(* CoDeSys 2.3 project: cy-162.pro *)
(* Title: cy-wg-24 - ClevergyAS *)
(* Author: Andrea Laini *)
(* Libraries: OSCAT\oscat_basic_333_pfc_2000.lib*20.4.16 13:29:42, mod_com.lib 16.5.13 14:00:50, SerComm.lib 16.5.13 14:00:50, Serial_Interface_01.lib 22.4.13 12:50:14, Modb_l05.lib*22.4.13 12:50:12, SysLibFile.lib 16.5.13 14:00:50, Util.lib 16.5.13 14:00:50, SYSLIBCALLBACK.LIB 16.5.13 14:00:50, SysLibRtc.lib 16.5.13 14:00:50, SysLibSockets.lib 22.5.14 16:16:32, SysLibEvent.lib 16.5.13 14:00:50, SysLibTime.lib 16.5.13 14:00:48, SysLibPlcCtrl.lib 16.5.13 14:00:50, SysLibStr.lib 16.5.13 14:00:50, Standard.lib 20.5.14 08:13:26, Iecsfc.lib 16.5.13 14:00:50 *)

(* PLC configuration (modules and I/O channels)
VPN_STATUS AT %IX0.0 [BOOLOnX_I] I 1: Digital Input
DI02 AT %IX0.1 [BOOLOnX_I] I 2: Digital Input
COORD_STATUS AT %IX0.2 [BOOLOnX_I] I 3: Digital Input
DI04 AT %IX0.3 [BOOLOnX_I] I 4: Digital Input
Modbus variables [PFC200MODBUS] node 1, in %IB0 out %QB0 {PlcStopBehaviour = 1; FiledbusErrorBehaviour = 1; TcpOperation = 0; TcpPort = 502; TcpTimeout = 600; UdpOperation = 0; UdpPort = 502; RtuOperation = 0; NodeId = 200; ResponseTimeout = 5000; Interface = 0; Baud = 38400; StopBits = 2; Parity = 0; FlowCtrl = 0; PhysInterface = 1}
Modbus-Master [MB_MASTER] node 2, in %IB0 out %QB0
*)

(* Global variable list: Global_Constants *)
VAR_GLOBAL CONSTANT

	Plant_NAME			: STRING :='cySN:162  cyVER:0 Q5904 via COMBONI Desenzano';
	Plant_SN				: DWORD  :=162;	  	(* S/N Impianto di telecontrollo *)
	Plant_SW_VER			: WORD   :=0;		(* Versione SW installata *)


	GEOLUMEN_COORD_VERSION:BYTE:=2;


	(* Plant-dependent constants *)
	LATITUDE 										: REAL:=45.45522;
	LONGITUDE										: REAL:=10.56686;
	ASTRO_TWILIGHT_MORNING_MODE					: BYTE:=0;
	ASTRO_TWILIGHT_EVENING_MODE					: BYTE:=0;
	COUNTRY_CODE 									: STRING:='IT';
	MAX_LUXNUM										: WORD := 1;
	MAX_GEOLUMENNODES								: WORD :=MAX_LUXNUM;
	MAX_LOG_ROW									: WORD :=2; (*MAX_LUXNUM	/10 +1 per eccesso*)
	MAX_RETRY_NO_FEEDBACK_GEOLUMEN_NODES			: WORD:=20;
	MAX_RETRY_STATUS_NOT_ALIGNED_GEOLUMEN_NODES       : WORD:=360;
	TIME_WAIT_RETRY_NOT_ALIGNED						: TIME:=T#10m;
	TIME_NO_FEEBACK_RESEND_STATUS					: TIME:=T#20m;

	(*tempi debug comandi global *)
	PRE_TIME_ENFORCE_GON 							: TIME:=T#10m;
	PRE_TIME_CLOSE_GOFF 								: TIME:=T#100m;
	TRIALS_ENFORCE_GON 								: WORD:=60;
	PERIOD_ENFORCE_GON 								: TIME:=T#1m;
	PERIOD_ENFORCE_GOFF 							: TIME:=T#15m;

	GEOLUMEN_SEND_TIME : TIME:=T#1s;

	(* Internal, tech const *)
	MAX_ARRAY_MSG	: BYTE:=250;
	ANALOG			: BOOL:=0;
	DIGITAL			: BOOL:=1;

	(* Filesystem *)
	FilesPath  			: STRING :='/media/sd/';
	MapConf_Path			: STRING :=	'/media/sd/';

	Luxlist_FileName	: STRING :='_LUX_LIST.txt';
	Cfg_FileName		: STRING :='CFG.txt';

	(* Colour Visu *)
	COLOR_RED			: DWORD 	:= 16#2020F0;
	COLOR_YELLOW		: DWORD	:= 16#20F0F0;
	COLOR_GREEN		: DWORD	:= 16#20F020;
	COLOR_GREEN_OFF	 : DWORD	:= 16#108010;

	(* TCP Logger *)
	Logger_SERVER		: STRING:='';
	Logger_IP				: STRING:='192.168.100.3';
	Logger_PORT			: WORD  :=80;
	Logger_GETSTART		: STRING:='GET /cygmsrv/hsgm.ashx?';
	Logger_GETEND		: STRING:='$R$N$R$N';
	Logger_CHECK			: STRING:='True';
	Logger_CRLF			: STRING:='$R$N';
	Logger_DataFile		: STRING:='/media/sd/LOG.DAT';
	Logger_DataFileOld	: STRING:='/media/sd/LOG.BCK';
	Logger_IndexFile	: STRING:='/media/sd/LOG.IDX';
	Logger_ConnRetries	: BYTE:=5;
	Logger_RecoverMsgs	: BYTE:=25;

	(* TCP Remote *)
	Remote_PORT			: WORD  :=10;
	Remote_WELCOME		: STRING:='Connected$R$N';
	Remote_OK			: STRING:='OK$R$N';
	Remote_ERROR		: STRING:='ERROR$R$N';

	(* TCP Sockets *)
	MAX_SEND_TCP_SERVER					 : DWORD:=6000;(*60000*)
	MAX_RECEIVE_TCP_SERVER				 : DWORD:=12000;
	MAX_RECEIVE_TCP_SERVER_SOCKET	 	 : DWORD:=6000;
	MAX_SEND_TCP_CLIENT					 : DWORD:=6000;(*15000*)
	MAX_RECEIVE_TCP_CLIENT				 : DWORD:=6000;
	MAX_RECEIVE_TCP_CLIENT_SOCKET		 : DWORD:=6000;
	MAX_RECEIVE_UDP_SERVER				 : INT  :=1472;
	MAX_RECEIVE_UDP_CLIENT				 : INT  :=1472;
	CONNECT_WATCHDOG_TIME				 : TIME :=t#10s;


END_VAR

(* Global variable list: Global_Retain *)
VAR_GLOBAL RETAIN PERSISTENT

	(* valori retain per i LUX objects*)
	GlobalWorkingtime		: ARRAY [1..MAX_LUXNUM] OF DWORD; (* [sec] Internal working time counter *)
	GlobalPowerOnCycles	: ARRAY [1..MAX_LUXNUM] OF WORD;	(*/DWORD;  *) (* Internal counter of power-on cycles *)
	GlobalEnergyCounter	: ARRAY [1..MAX_LUXNUM] OF WORD; (* DWORD;  *) (* [E-1 kWh] Internal energy counter *)
	GlobalEnergyCounter_t 	: ARRAY [1..MAX_LUXNUM] OF DWORD; (* Temporary energy in E-2*Wsec *)

	(*configurazione degli astro *)
	ASTR_CONFIG   : ARRAY [1..MAX_LUXNUM] OF  type_ASTR_config;

	USE_RETAIN:BOOL:=FALSE;

	DEBUG_NO_CONTROL_LIGHTS : BOOL :=FALSE;
	DEBUG_SERIAL:BOOL:=FALSE;
	DEBUG_SAVE_SNAPSHOT:BOOL:=TRUE;
	USING_EXTERNAL_ASTRO:BOOL:=TRUE;

END_VAR

(* Global variable list: Global_Variables *)
VAR_GLOBAL

	SYS    : typ_SYS;
	Logger : typ_Logger;

	LAMP : LAMP_AL_GENERALE;

	PLC_ID				: STRING:='1' ; (* Identificativo del plc - interno al file cfg.txt  *)
	PLC_START_TIME 		:DT;

	SyncLogRequest: BOOL:=FALSE;
	TimerLogLux : ARRAY[1..MAX_LOG_ROW] OF TON;
	TimerLogLuxSync : ARRAY[1..MAX_LOG_ROW] OF TON;
	TimerLogLuxSyncDone : ARRAY[1..MAX_LOG_ROW] OF BOOL;
	TimingLuxBase : TIME;
	logRowLux:INT:=0;
	IS_PRE_GLOBAL_ON_ONGOING:BOOL:=FALSE;

	(*contSts0:DWORD:=0;
	contSts1:DWORD:=0;*)
	warningHFileLogSend:BOOL:=FALSE;

	(*Tabella della lista dei lux GEOLUMEN costruita sulla base del file di configurazione*)
	TabListLux : ARRAY [1..MAX_LUXNUM] OF type_TabListLuxGeolumen;
	TabListLuxSendAuth : ARRAY [1..MAX_LUXNUM]  OF WORD:=0;

	LuxElement		: ARRAY [1..MAX_LUXNUM] OF obj_LUX:=(CTRL_MODE:=2,CTRL_MODE_BackUp:=2); (* Lista di variabili Lux   *)
	LuxGeolumenChangeFlag : ARRAY [1..MAX_LUXNUM] OF INT;

	TimerLogAstro : ARRAY[1..MAX_LOG_ROW] OF TON;
	TimerLogAstroSync : ARRAY[1..MAX_LOG_ROW] OF TON;
	TimerLogAstroSyncDone : ARRAY[1..MAX_LOG_ROW] OF BOOL;
	TimingAstroBase : TIME;
	tIndex:INT;
	logRowAstro:INT:=0;
	isGeolumenNodesOffDuringDay:isGeolumenNodesOffDuringDay;
	tmpBoolGoffDay:BOOL;

	GeolumenNodeList	:GeolumenNodeList;

	(* Astro crono *)
	ASTR   			: ARRAY [1..MAX_LUXNUM] OF obj_ASTR;
	astroGen			 : obj_ASTR;
	CronEd : obj_CRON_EDITOR:=(crono_type:='ASTR');

	(*Lux *)
	MsgRecBuffer	: ARRAY[0..MAX_ARRAY_MSG ] OF type_MsgReceive; (*Array contenente i messaggi in arrivo e gestito in modo circolare*)
	KEYON :BOOL;

	LuxGeolumenNodes : ARRAY [1..MAX_LUXNUM] OF obj_GeolumenNode:=(MAX_RETRY_NO_FEEDBACK:=MAX_RETRY_NO_FEEDBACK_GEOLUMEN_NODES,
															MAX_RETRY_STATUS_NOT_ALIGNED:=MAX_RETRY_STATUS_NOT_ALIGNED_GEOLUMEN_NODES);

	LuxGeolumenNodesAlignFlags : ARRAY [1..MAX_LUXNUM] OF BOOL:=FALSE;
	LuxGeolumenNodesCurrent : ARRAY [1..MAX_LUXNUM] OF DWORD;
	Missing : ARRAY [1..MAX_LUXNUM] OF BOOL:=FALSE;
	missingCount:INT:=0;

	(*Geolumen rs232 dependent*)
	COM0:SERIAL_INTERFACE := (xOPEN_COM_PORT := TRUE, bCOM_PORT_NR  := 0, cbsBYTESIZE := BS_8,
							cbBAUDRATE := BAUD_115200, cpPARITY := PARITY_NO, csSTOPBITS := STOPBITS_1, cfFLOW_CONTROL := NO_FLOW_CONTROL);
	ReceiveBuffer:typRing_Buffer;
	xCoupledAll		:BOOL;
	obj_GeolumenCoordinator:obj_GeolumenCoordinator;
	LuxGeolumenDiagnostics:LuxGeolumenDiagnostics;
	SendDataQueue:SendDataQueue;

END_VAR

(* Data type in DT_LUX *)
TYPE en_ActionKey :
(
	NormalMode 	:= 0,
	SwitchON		:= 1,
	SwitchOFF		:= 2,
	Restore			:= 3
);
END_TYPE

(* Data type in DT_LUX *)
TYPE en_KeyMode :
(
	BUTTON_NO		:=01,
	BUTTON_NC		:=02,
	SWITCH_NO		:=03,
	SWITCH_NC			:=04
);
END_TYPE

(* Data type in DT_Logger *)
TYPE en_Logger_ErrLev :
(
	EL_Log			:=0,
	EL_Wrn			:=1,
	EL_Alarm		:=2,
	EL_AlarmStop	:=3,

	EL_Evt			:=4
);
END_TYPE

(* Data type in DT_Logger *)
TYPE en_Logger_Status :
(
	S_Logger_UNKNOWN := 0,
	S_Logger_IDLE,
	S_Logger_WAITCONN,
	S_Logger_WAITTX,
	S_Logger_WAITRESP,
	S_Logger_ERROR
);
END_TYPE

(* Data type in DT_LUX *)
TYPE en_Modality :
(
	ManualeOff 	:= 0,
	ManualeOn 	:= 1,
	Cronografo	:= 2,
	Timer		:= 3,
	KeyControl	:= 4
);
END_TYPE

(* Data type in System *)
TYPE en_MsgType :
(
	COMPLETED:=0, (*Il messaggio è stato elaborato*)
	REQAUTH0:= 1,  (*Richiesta in corso a cui rispondere*)
	REQAUTH1:=2,  (*Nodo già acquisito in rete*)
	DATAREC:=3,
	ECHO:=4,
	NODE_DELETED:=5,
	MED:=6
);
END_TYPE

(* Data type in System *)
TYPE en_StartingState :
(
	NOT_AUTHORISE  := 0,
	READ_NODE
);
END_TYPE

(* Data type in DT_SYS *)
TYPE en_SYS_Objects :
(
	EO_SYS		:=0,  (* PLC *)
	EO_VPN		:=1,  (* VPN *)
	EO_DOOR	:=2,  (* Door & access control *)

	EO_CAL		:=10, (* Caldaia *)
	EO_CIR		:=11, (* Circolatore *)
	EO_CRON		:=12, (* Crono-termostato *)
	EO_VRD		:=13, (* Valvola miscelatore pannelli *)
	EO_CTL		:=14, (* Contalitri *)
	EO_CTB		:=15, (* Contabilizzatore *)
	EO_TPV		:=16, (* Temperature probes values *)
	EO_PPV		:=17, (* Pressure probes values *)
	EO_PBV		:=18, (* Over-Pressure Alarms *)
	EO_TBV		:=19, (* Over-Temperature Alarms *)
	EO_PMV		:=20, (* Under-Pressure Alarms *)
	EO_GRU		:=21, (* Gruppo termico *)
	EO_PDC		:=22, (* Pompa di calore *)
	EO_SOL		:=23, (* Pannello solare termico *)
	EO_ESOL		:=24, (* Pannello solare fotovoltaico *)
	EO_GAS		:=25, (* Contatore GAS *)
	EO_PORT		:=26, (* Misuratore di portata *)
	EO_FPV		:=27, (* Flow probes values *)
	EO_ANZ		:=28, (* Analizzatore di rete *)
	EO_SCA		:=29, (* Signal Control Alarms *)
	EO_LUX		:=30, (* Illumination point *)
	EO_LUXM		:=31, (* Metered illumination point*)
	EO_PSG		:=32, (* Sensore di passaggio *)
	EO_HVAC		:=33, (*Heating, Ventilating and Air Conditioning*)
	EO_HYGRV	:=34, (*Valori sensori di umidità relativa (0.1%)*)
	EO_COOV		:=35, (*Valori sensori CO2 (PPM)*)

	EO_ASTR		 :=46, (*Astro crono *)




	EO_ZGW			:=200,  (* ZigBee - Gateway *)
	EO_ZRM			:=201,	(* ZigBee - Repeater *)
	EO_ZREL			:=202,	(* ZigBee - Actuator rele *)
	EO_ZTHL			:=203,	(* ZigBee - Temperature Sensor *)

	EO_ASGW			:=250,	(* ASi - Gateway *)
	EO_ASCBI			:=251,	(* ASi - Input Board, Ciabatta *)

	EO_LON				:=1000, (* Bus - LON *)
	EO_MODBUS			:=1001, (* Bus - MODBUS *)
	EO_MBUS				:=1002, (* Bus - M-BUS *)
	EO_MODBUS_TCP	:=1003, (* Bus - MODBUS TCP *)

	EO_GENERIC			:=9000, (* Generic dataset *)
	EO_EXPO				:=9001 (* EXPO dataset *)
);
END_TYPE

(* Data type in DT_SYS *)
TYPE en_SYS_Status :
(
	S_UNKNOWN  := 0,
	S_STARTUP,
	S_INIT_RTC,
	S_INIT_VAR,
	S_AUTOTEST,
	S_RUNNING,
	S_SHUTDOWN,
	S_HALT,
	S_RELOAD,
	S_STARTER
);
END_TYPE

(* Data type in DT_SYS *)
TYPE typ_Condition :
STRUCT
	Enable		:	BYTE;	(*	0: Condition event not used		(disable condition event)
								1: Boolean event: trig On	(rele, switch, sensors digital input..)
								2:    ''    ''  : trig Off		
								3:	  ''    ''  : trig On/Off
								4: Tod event: trig On		(Time of day)
								5: Tod event: trig Off		(Trig On/Off not expected -> it's a schedule! )
							 *)

	(* Boolean event *)
	OnIN		:	BOOL;	(* Input event generating an On *)
	OffIN		:	BOOL;	(* Input event generating an Off  *)

	OnValue		:	BOOL;	(* Value to trig an On *)
	OffValue	:	BOOL;	(*   ''        ''   Off	 *)


	(* Time of the day event (absolute time) *)
	OnTime		:	TOD;	(* Time at which trig an On (hh:mm) *)
	OffTime		:	TOD;	(*  ''            ''     Off (hh:mm)  *)


END_STRUCT
END_TYPE

(* Data type in DT_CRON *)
TYPE typ_Cron_Calendar :
STRUCT
	Profile		: ARRAY[0..384] OF BYTE;
END_STRUCT
END_TYPE

(* Data type in DT_CRON *)
TYPE typ_Cron_Jolly :
STRUCT
	Start		: DT;
	End			: DT;
	Temp		: WORD;
	Flags		: WORD; (* B0:Enabled B1..B15:Unused *)
END_STRUCT
END_TYPE

(* Data type in DT_CRON *)
TYPE typ_Cron_Profile :
STRUCT
	Flags		: WORD;
	Setpoint	: ARRAY [0..95] OF WORD;
END_STRUCT
END_TYPE

(* Data type in DT_Logger *)
TYPE typ_Logger :
STRUCT
	Status		: en_Logger_Status;

	SendReq		: BOOL;
	SendIdx		: DWORD;
	SendData	: ARRAY [0..MAX_SEND_TCP_CLIENT] OF BYTE;
	SendLen		: DINT;

	TData		: ARRAY [0..MAX_SEND_TCP_CLIENT] OF BYTE;
	TLen		: DINT;

	LastIdxPos	: DWORD;

	(* Temporary variables used by objects *)
	s1			: STRING(256);
	i1			: WORD;

END_STRUCT
END_TYPE

(* Data type in DT_SYS *)
TYPE typ_SYS :
STRUCT
	Status			: en_SYS_Status;
	Warning		: BOOL;
	Alarm			: BOOL;
	AlarmStop		: BOOL;

	Time_LogString	: STRING(255);
	Time_Year		: WORD;
	Time_Month		: BYTE;
	Time_Day		: BYTE;
	Time_Hour		: BYTE;
	Time_Min		: BYTE;

	Time_CT_DT		: DT;
	Time_CT_Day		: WORD;
	Time_CT_Quarter	: BYTE;

	LastLogs_Idx	: BYTE;
	LastLogs_Dat	: ARRAY[0..5] OF STRING(255);
	LastLogs_Msg	: ARRAY[0..5] OF STRING(255);

END_STRUCT
END_TYPE

(* Data type *)
TYPE type_ASTR_config :
STRUCT
	id:DWORD;
	twilightMorningMode:BYTE;
	twilightEveningMode:BYTE;
	preSunrise:BYTE;
	postSunrise:BYTE;
	preSunset:BYTE;
	postSunset:BYTE;
END_STRUCT
END_TYPE

(* Data type in DT_LUX *)
(* La seguente struttura ha la funzione di collegare l'id del lux con i relativi dati qui indicati *)
(* In tal modo la visualizzazione dello stato dei lux viene eseguita associando l'ID dell'array contenente questa struttura*)

TYPE type_DataLuxForVis :
STRUCT
	VisStatus	: DWORD; (* valori di status_vis   *)
	VisTimer	: TIME;	(* Valori dei timer  *)
	VisMod		: en_Modality; (* Impostazione mode  *)
END_STRUCT
END_TYPE

(* Data type in DT_LUX_GEOLUMEN *)
TYPE type_LuxGeolumenStatus :
STRUCT
	ID_Geolumen: DWORD;
	DimmValue_0 : WORD;
	DimmValue_1 : WORD;
	DimmValue_2 : WORD;
	LampCurrent:DWORD;LampPower:DWORD;LampVoltage:DWORD;
	lqiLast, lqiAvg, lqiMax, lqiMin:WORD;
	lastPar:STRING(255);
END_STRUCT
END_TYPE

(* Data type in DT_LUX *)
TYPE type_LuxOutput :
STRUCT
	DigitalOut	:	BOOL;
	AnalogOut	:	WORD;
	TypeOut	:	BOOL;
END_STRUCT
END_TYPE

(* Data type in System *)
TYPE type_MsgReceive :
STRUCT
	Msg		:STRING (255);
	MsgType	: en_MsgType; (*Indica il tipo di messaggio STS0, STS1,...*)
	dwMacAdd	: DWORD;

END_STRUCT
END_TYPE

(* Data type in DT_LUX *)
(* Struttura utile per la lista dei lux *)

TYPE type_TabListLux :
STRUCT
	LuxNumber: WORD;
	MODE: WORD;
	MacAdd: DWORD;
	MacAddH: WORD;
	MacAddL: WORD;
	StMacAdd	: STRING(8);
END_STRUCT
END_TYPE

(* Data type in DT_LUX_GEOLUMEN *)
(* Struttura utile per la lista dei lux *)

TYPE type_TabListLuxGeolumen :
STRUCT
	LuxNumber	: DWORD;
	LuxID_Geolumen		: DWORD;
	MacAdd	: DWORD;
	MacAddH	: WORD;
	MacAddL	: WORD;
	StMacAdd	: STRING(8);
	xCoupled	: BOOL;
END_STRUCT
END_TYPE

(* POU PLC_PRG, ST *)
PROGRAM PLC_PRG
VAR CONSTANT
	TIME_LUX_LOG_NORMAL:TIME:=T#5m;
	TIME_ASTRO_LOG_NORMAL:TIME:=T#30m;
	TIME_LUX_PROC:TIME:=T#200ms;
	TIME_STATUS_2:TIME:=T#180M;
END_VAR
VAR
	DAILY_RESET_DONE:BOOL;
	TimerLux:TON;
	Timer1: TON;  (*Fast controls tick *)
  	Timer2: TON; (* Plant control tick *)
	TimerSnapshot:TON;
	maxLoggerRow:INT;
	TimerAstroQuadroNotte:TON;
	TimerAstroQuadroGiorno:TON;
	contaSera:INT:=0;
	contaMattina:INT:=0;

	xOpenPort		: BOOL := TRUE;
	xInitPort			: BOOL;
	xSendActive	: BOOL;
	SendString		: STRING(255) := 'CMD_AUTHORISE=0';
	xStartSend		: BOOL;

	GeoNodeIndex:INT:=1;
	i :INT :=1;
	LuxCount	: WORD:=1;
	ValInCrono	: INT; (* Valore del setpoint del crono *)
	counter		: WORD;
	tmpIndex:INT;

	tmpMaxEvening:BYTE;
	tmpMinEvening:BYTE;
	tmpMinMorning:BYTE;
	tmpMinPreEvening:BYTE;
	tmpMaxPreEvening:BYTE;
	tmpMaxPostEvening:BYTE;
	tmpMinPostEvening:BYTE;
	tmpMinPreMorning:BYTE;
	tmpMaxPostMorning:BYTE;
	tmpTime:TIME;


END_VAR
(*
	Network setup:
		IP  = 192.168.100.2 | MSK = 255.255.255.0
		GW	= 192.168.100.1 | DNS = 192.168.100.1
		SNTP = 193.204.114.232 (3600s) ==> 192.168.100.3
*)


(*==============================*)
(*=====    Main control machine    ====*)
(*==============================*)

MainCtrl();

Logger_Proc();

Remote_Proc();
END_PROGRAM
ACTION MainCtrl:
CASE Sys.Status OF

	(* stato STARTUP
	     - carico la lista dei nodi Geolumen da accettare (ID palo, MAC)
	     - apro la porta seriale
	     - invio al coordinatore Geolumen il comando CMD_AUTHORISE=0
	*)
	S_STARTUP:

		DAILY_RESET_DONE:=FALSE;

		(* pongo a zero valore variabili essenziali*)
		FOR counter := 1 TO MAX_LUXNUM DO
			TabListLux[counter].LuxID_Geolumen:=0;
			TabListLux[counter].MacAdd:=0;
			TabListLux[counter].MacAddH:=0;
			TabListLux[counter].MacAddL:=0;
			TabListLux[counter].StMacAdd:='';
			TabListLux[counter].LuxNumber:=0;
			TabListLux[counter].xCoupled:=FALSE;
			LuxElement[counter].ID:=0;
			ASTR[counter].ID:=0;
			LuxGeolumenNodes[counter].ID_Lux:=0;
			LuxGeolumenNodes[counter].ID_Geolumen:=0;
		END_FOR

		(* caricamento lista nodi *)
		GeolumenNodeList();

		(* apro la porta seriale *)
		xSendActive:=FALSE;
		COM0((*	bCOM_PORT_NR 	:= 0,
				cbBAUDRATE     	 := BAUD_38400,
			(*	cbBAUDRATE 		:= wBaudRate, *)
				cbsBYTESIZE		:= BS_8,  (*bDataBits,*)
				cpPARITY			:= PARITY_NO, (* bParity,*)
				csSTOPBITS		:= STOPBITS_1,
				cfFLOW_CONTROL	:= NO_FLOW_CONTROL,	(*bFlowControl,			*) *)
				cbBAUDRATE     	 := BAUD_115200,
				utRECEIVE_BUFFER := ReceiveBuffer,
				ptSEND_BUFFER	:= ADR(SendString),
				xINIT				:=  xInitPort,
		     		xOPEN_COM_PORT 	:= TRUE,	(*xOpenPort,*)
				iBYTES_TO_SEND	:= LEN(SendString)+1,
				xSTART_SEND		:= xSendActive );

		(*proseguo con lo stato successivo sse porta seriale aperta *)
		IF COM0.xCOM_PORT_IS_OPEN THEN
			Sys.Status:=S_INIT_RTC;

			(* anzitutto blocco auto-auth da parte dei nodi*)
			obj_GeolumenCoordinator.blockNodeAutoAdd();

		END_IF

	(* stato INIT_RTC
	     - init RTC PLC
	     - sync time coordinatore Geolumen
	*)
	S_INIT_RTC:

		(* aggiorno stringhe RTC as usual*)
		RTC_Update();

		(* aggiorno ora del coordinatore con la mia e proseguo allo stato successivo come al solito *)
		IF Sys.Time_Year>2000 THEN
			obj_GeolumenCoordinator.updateNetworkTime();
			Sys.Status:=S_INIT_VAR;
		END_IF

	(* stato S_INIT_VAR
	     - init variabili oggetti
	*)
	S_INIT_VAR:

		(*tutti i LUX presenti sono di default e ad ogni riavvio di tipo dimming e di modo 2 - Cronografo *)
		FOR counter := 1 TO MAX_LUXNUM DO
			LuxElement[counter].DimmingType:=1;
			LuxElement[counter].CTRL_MODE := 2 ; (* TabDefaultLux[counter].Mode; //copio il mode nella tabella delle variabili dei lux 	*)
			LuxElement[counter].CTRL_MODE_backUp := 2;  (* TabDefaultLux[counter].Mode; //salvo il mode di backup per il ripristina modo	*)
		END_FOR

		(*ripeto il comando di esclusione di accesso da parte dei nodi, per sicurezza*)
		obj_GeolumenCoordinator.blockNodeAutoAdd();


		(* definizione ASTRO di quadro, per test *)
		tmpMinEvening:=100;
		tmpMaxEvening:=0;
		tmpMinMorning:=100;
		tmpMinPreEvening:=30;
		tmpMaxPreEvening:=0;
		tmpMaxPostEvening:=0;
		tmpMinPostEvening:=100;
		tmpMinPreMorning:=30;
		tmpMaxPostMorning:=0;

		(* inizializzo gli astro con eventale stato retain *)
		FOR i:=1 TO MAX_LUXNUM DO
			ASTR[i].ID:=ASTR_CONFIG[i].ID;
			ASTR[i].rLatitude:=LATITUDE;
			ASTR[i].rLongitude:=LONGITUDE;
			ASTR[i].countryCode:=COUNTRY_CODE;
			IF(USE_RETAIN=FALSE) THEN
				ASTR[i].twilightEveningMode :=ASTRO_TWILIGHT_EVENING_MODE;
				ASTR[i].twilightMorningMode :=ASTRO_TWILIGHT_MORNING_MODE;
				ASTR_CONFIG[i].preSunrise:=ASTR[i].preSunrise;
				ASTR_CONFIG[i].postSunrise:=ASTR[i].postSunrise;
				ASTR_CONFIG[i].preSunset:=ASTR[i].preSunset;
				ASTR_CONFIG[i].postSunset:=ASTR[i].postSunset;
				ASTR_CONFIG[i].twilightEveningMode:=ASTR[i].twilightEveningMode;
				ASTR_CONFIG[i].twilightMorningMode:=ASTR[i].twilightMorningMode;
			ELSE
				ASTR[i].preSunrise:=ASTR_CONFIG[i].preSunrise;
				ASTR[i].postSunrise:=ASTR_CONFIG[i].postSunrise;
				ASTR[i].preSunset:=ASTR_CONFIG[i].preSunset;
				ASTR[i].postSunset:=ASTR_CONFIG[i].postSunset;
				ASTR[i].twilightEveningMode:=ASTR_CONFIG[i].twilightEveningMode;
				ASTR[i].twilightMorningMode:=ASTR_CONFIG[i].twilightMorningMode;
			END_IF


			IF ASTR[i].twilightEveningMode < tmpMinEvening THEN tmpMinEvening:=ASTR[i].twilightEveningMode; END_IF
			IF ASTR[i].twilightMorningMode < tmpMinMorning THEN tmpMinMorning:=ASTR[i].twilightMorningMode; END_IF
			IF ASTR[i].preSunset > tmpMinPreEvening THEN tmpMaxPreEvening:=ASTR[i].preSunset; END_IF
			IF ASTR[i].postSunset < tmpMinPostEvening THEN tmpMinPostEvening:=ASTR[i].postSunset; END_IF
			IF ASTR[i].preSunrise < tmpMinPreMorning THEN tmpMinPreMorning:=ASTR[i].preSunrise; END_IF
			IF ASTR[i].postSunrise > tmpMaxPostMorning THEN tmpMaxPostMorning:=ASTR[i].postSunrise; END_IF

		END_FOR

		astroGen.ID:=1;
		astroGen.rLatitude:=LATITUDE;
		astroGen.rLongitude:=LONGITUDE;
		astroGen.countryCode:=COUNTRY_CODE;
		astroGen.twilightEveningMode:=tmpMinEvening;
		astroGen.twilightMorningMode:=tmpMinMorning;
		astroGen.preSunset:= tmpMaxPreEvening;
		astroGen.postSunset:= tmpMinPostEvening;
		astroGen.preSunrise:= tmpMinPreMorning;
		astroGen.postSunrise:=tmpMaxPostMorning;

		(*chiedo agli eventuali nodi geoluem connesso il loro stato*)
		SendDataQueue(pTxData:=ADR(obj_GeolumenCoordinator.getStatusAllFeedback));
		SendDataQueue.addMessage();

		(*recall lux*)
		obj_GeolumenCoordinator.luxRecall();


		(*procedo con stato successivo *)
		Sys.Status:=S_STARTER;

	(* stato S_STARTER
	     - ad oggi logga solo avvio
	*)
	S_STARTER:
		LogEv(EL_Wrn,EO_SYS,0,1,CONCAT('System_startup_v',WORD_TO_STRING(Plant_SW_VER)));
		Sys.Status:=S_RUNNING;
		PLC_START_TIME:=SYS.Time_CT_DT;

	(* stato S_RUNNING
	     - aggiorna lo stato di ASTR e di LUX
	     - si occupa di mantenere la corrispondenza di stato tra LUX e GEOLUMENNODE
	*)
	S_RUNNING:

		(*salvo stato nodi su sd, ogni ora *)
		TimerSnapshot(IN:=NOT TimerSnapshot.Q,PT:=T#1h);
		IF DEBUG_SAVE_SNAPSHOT AND TimerSnapshot.Q THEN
			GeolumenSaveNodeStatus();
		END_IF

		(*aggiorni eventi SCA e SYS as usual*)
		Timer1(IN:=NOT Timer1.Q,PT:=T#50ms);
		IF Timer1.Q THEN
			(* Update meters *)
			SCA_Proc();
			(* Update system checks *)
			SYS_Proc();
		END_IF

		(*aggiorno stringhe RTC as usual*)
		Timer2(IN:=NOT Timer2.Q,PT:=T#500ms);
		IF Timer2.Q THEN
			(* Read current date/time *)
			RTC_Update();
			(*per PIANO C*)
			isGeolumenNodesOffDuringDay(isGeolumenNodesOffDuringDay=>tmpBoolGoffDay);
		END_IF

		(* gestione astr di quadro per eventuali comandi global di enforcing e gestione PIANO C*)
		(* + reset coordinatore prima di accensione serale*)
		AstroGen(localTime:=Sys.Time_CT_DT);
		IF(SYS.Time_CT_DT>=AstroGen.timeStart-PRE_TIME_ENFORCE_GON AND SYS.Time_CT_DT<AstroGen.timeStart) THEN
			IS_PRE_GLOBAL_ON_ONGOING:=TRUE;

			FOR GeoNodeIndex:=1 TO MAX_LUXNUM  DO
				IF LuxElement[GeoNodeIndex].ID <> 0 THEN
					LuxGeolumenNodes[GeoNodeIndex].resetLampIndicators();
				END_IF
			END_FOR

		ELSE
			IS_PRE_GLOBAL_ON_ONGOING:=FALSE;
			DAILY_RESET_DONE:=FALSE;
		END_IF


		IF(IS_PRE_GLOBAL_ON_ONGOING AND DAILY_RESET_DONE=FALSE) THEN
			(*LuxGeolumenDiagnostics.executeCommandReset();*)
			DAILY_RESET_DONE:=TRUE;
		END_IF


		(* gestione con global, debug and test *)
		(*TimerAstroQuadroNotte(IN:=NOT TimerAstroQuadroNotte.Q,PT:=PERIOD_ENFORCE_GON);
		(* la sera lancio un set iniziale di Global a 100 *)
		IF(SYS.Time_CT_DT>=AstroGen.timeStart-PRE_TIME_ENFORCE_GON AND TimerAstroQuadroNotte.Q AND contaSera<TRIALS_ENFORCE_GON ) THEN
			(*obj_GeolumenCoordinator.sendGlobalON();*)(*DIEGO REMOVE*)
			contaSera:=contaSera+1;
			contaMattina:=0;
		ELSIF contaSera>=TRIALS_ENFORCE_GON  THEN
			contaMattina:=0;
		END_IF

		TimerAstroQuadroGiorno(IN:=NOT TimerAstroQuadroGiorno.Q,PT:=PERIOD_ENFORCE_GOFF);
		IF(SYS.Time_CT_DT>=AstroGen.timeEnd AND SYS.Time_CT_DT<AstroGen.timeStart-PRE_TIME_CLOSE_GOFF AND TimerAstroQuadroGiorno.Q) THEN
			(*obj_GeolumenCoordinator.sendGlobalOFF();*)(*DIEGO REMOVE*)
			contaSera:=0;
			contaMattina:=contaMattina+1;
		END_IF*)

		(* eseguo CronEd *)
		CronEd();

		(* eseguo oggetto di diagnostica per comandi via PLC Web Visu *)
		LuxGeolumenDiagnostics();

		(* eseguo ciclo transfer data and parse *)
		obj_GeolumenCoordinator(ReceiveBufferPtr:=ADR(ReceiveBuffer),MsgRecBufferPtr:=ADR(MsgRecBuffer));

		(* eseguo aggiornamento stato lux e verifica coerenza stato desiderato e stato effettivo*)
		(* i lux sono considerati in sequenza ogni TIME_LUX_PROC*)
		(*TimerLux(IN:=NOT TimerLux.Q, PT:=TIME_LUX_PROC);
		IF TimerLux.Q THEN*)

			IF  LuxElement[LuxCount].ID <> 0  THEN (* esegue scansione dei lux dell'impianto solo se presenti *)

				(* salvo lo stato desiderato corrente del LuxGeolumenNode *)
				LuxGeolumenChangeFlag[LuxCount]:=LuxGeolumenNodes[LuxCount].desideredDimmValue;

				CASE LuxElement[LuxCount].CTRL_MODE OF
					(*
					0:
					1:	 *)
					2:
						IF  ASTR[LuxCount].ID <> 0 THEN
							(* se il mode è settato come cronografo gestisco accensione a orologio *)
							ASTR[LuxCount]( localTime:=Sys.Time_CT_DT,SetPoint=>ValInCrono);
							LuxElement[LuxCount](	ValInCronoInLux:=ValInCrono/10, (* astr 0-100, Lux 0-100 *)
										       		LuxAnalogOut => LuxGeolumenNodes[LuxCount].desideredDimmValue,
									 	       		WorkingTime:=GlobalWorkingtime[LuxCount],
										       		PowerOnCycles:=GlobalPowerOnCycles[LuxCount],
												EnergyCounter:=GlobalEnergyCounter[LuxCount],
										    	   	EnergyCounter_t:=GlobalEnergyCounter_t[LuxCount],KeyQty:=2);
						END_IF


				END_CASE


				LuxElement[LuxCount](	LuxAnalogOut => LuxGeolumenNodes[LuxCount].desideredDimmValue,
									WorkingTime:=GlobalWorkingtime[LuxCount],
									PowerOnCycles:=GlobalPowerOnCycles[LuxCount],
									EnergyCounter:=GlobalEnergyCounter[LuxCount],
									EnergyCounter_t:=GlobalEnergyCounter_t[LuxCount],KeyQty:=2);  (*, KeyMode:=KeyTest.KeyMode); *)


				(* aggiorno lo stato desiderato del LUX GeolumenNode*)
				LuxGeolumenNodes[LuxCount].updateDesideredState();

				(* se è diverso dal precedente, invio richiesta modifica stato *)
				IF(isCoordinatorBooted() AND LuxGeolumenChangeFlag[LuxCount]<>LuxGeolumenNodes[LuxCount].desideredDimmValue) THEN
					(*resetto i contatori di eventuale disallineamento*)
					LuxGeolumenNodes[LuxCount].resetRetryCounters();

					(*in modalitò Crono e piano C non mando mai spegnimento *)
					IF  LuxGeolumenNodes[LuxCount].ID_Geolumen <>0 AND
					     NOT DEBUG_NO_CONTROL_LIGHTS AND
					     NOT (LuxElement[LuxCount].CTRL_MODE = 2 AND USING_EXTERNAL_ASTRO=TRUE AND LuxGeolumenNodes[LuxCount].desideredDimmValue=0)  THEN
						(*invio set*)
						SendDataQueue(pTxData:=ADR(LuxGeolumenNodes[LuxCount].toSendSetString));
						SendDataQueue.addMessage();
					END_IF

				END_IF

				(*aggiorno controllo stato dei nodi *)
				LuxGeolumenNodes[LuxCount].checkStatusANDPresence();
				LuxGeolumenNodesAlignFlags[LuxCount]:=isGeolumenEqualStatus(LuxGeolumenNodes[LuxCount].desideredState, LuxGeolumenNodes[LuxCount].feedbackState);

				(*rettifico lo stato nel caso di modalità piano C *)

				IF USING_EXTERNAL_ASTRO AND tmpBoolGoffDay THEN

					LuxElement[LuxCount](Lux_State:=FALSE,
								Lux_StateAnalog:=0,
								WorkingTime:=GlobalWorkingtime[LuxCount],
								PowerOnCycles:=GlobalPowerOnCycles[LuxCount],
								EnergyCounter:=GlobalEnergyCounter[LuxCount],
								EnergyCounter_t:=GlobalEnergyCounter_t[LuxCount],KeyQty:=2);

					LuxGeolumenNodes[LuxCount].feedbackState.DimmValue_0:=0;
					LuxGeolumenNodes[LuxCount].feedbackState.DimmValue_1:=0;
					LuxGeolumenNodes[LuxCount].feedbackState.DimmValue_2:=0;

				END_IF

				(*regole statusLog*)
				IF USING_EXTERNAL_ASTRO AND tmpBoolGoffDay THEN
					LuxElement[LuxCount](WorkingTime:=GlobalWorkingtime[LuxCount],
									       PowerOnCycles:=GlobalPowerOnCycles[LuxCount],
									       EnergyCounter:=GlobalEnergyCounter[LuxCount],
									       EnergyCounter_t:=GlobalEnergyCounter_t[LuxCount]);
				ELSE
					IF luxGeolumenNodes[LuxCount].lampBroken AND Sys.Time_CT_DT-LuxGeolumenNodes[LuxCount].lastSeen>TIME_STATUS_2 THEN

								LuxElement[LuxCount](WorkingTime:=GlobalWorkingtime[LuxCount],
								PowerOnCycles:=GlobalPowerOnCycles[LuxCount],
								EnergyCounter:=GlobalEnergyCounter[LuxCount],
								EnergyCounter_t:=GlobalEnergyCounter_t[LuxCount],
								Status_Log:=-3);

					ELSIF luxGeolumenNodes[LuxCount].lampBroken AND (LuxGeolumenChangeFlag[LuxCount]<>LuxGeolumenNodes[LuxCount].desideredDimmValue) THEN

								LuxElement[LuxCount](WorkingTime:=GlobalWorkingtime[LuxCount],
								PowerOnCycles:=GlobalPowerOnCycles[LuxCount],
								EnergyCounter:=GlobalEnergyCounter[LuxCount],
								EnergyCounter_t:=GlobalEnergyCounter_t[LuxCount],
								Status_Log:=-1);


					ELSIF luxGeolumenNodes[LuxCount].lampBroken THEN

								LuxElement[LuxCount](WorkingTime:=GlobalWorkingtime[LuxCount],
								PowerOnCycles:=GlobalPowerOnCycles[LuxCount],
								EnergyCounter:=GlobalEnergyCounter[LuxCount],
								EnergyCounter_t:=GlobalEnergyCounter_t[LuxCount],
								Status_Log:=2);

					ELSIF  Sys.Time_CT_DT-LuxGeolumenNodes[LuxCount].lastSeen>TIME_STATUS_2 THEN
						LuxElement[LuxCount](WorkingTime:=GlobalWorkingtime[LuxCount],
								PowerOnCycles:=GlobalPowerOnCycles[LuxCount],
								EnergyCounter:=GlobalEnergyCounter[LuxCount],
								EnergyCounter_t:=GlobalEnergyCounter_t[LuxCount],
								Status_Log:=-2);
					ELSE
						LuxElement[LuxCount](WorkingTime:=GlobalWorkingtime[LuxCount],
								PowerOnCycles:=GlobalPowerOnCycles[LuxCount],
								EnergyCounter:=GlobalEnergyCounter[LuxCount],
								EnergyCounter_t:=GlobalEnergyCounter_t[LuxCount],
								Status_Log:=BOOL_TO_BYTE(LuxGeolumenChangeFlag[LuxCount]<>LuxGeolumenNodes[LuxCount].desideredDimmValue));
					END_IF
				END_IF


			END_IF



		(*END_IF*)

		LuxCount:=LuxCount+1;

		(*riparto dal primo se lux  finiti *)
		IF LuxCount > MAX_LUXNUM THEN LuxCount:=1; END_IF

		(*faccio comunque un check istantaneo di tutti i nodi, cosi da aggiornare e verificare  timer interno *)
		FOR GeoNodeIndex:=1 TO MAX_LUXNUM  DO
			IF LuxElement[GeoNodeIndex].ID <> 0 THEN
				LuxElement[GeoNodeIndex](
								WorkingTime:=GlobalWorkingtime[GeoNodeIndex],
								PowerOnCycles:=GlobalPowerOnCycles[GeoNodeIndex],
								EnergyCounter:=GlobalEnergyCounter[GeoNodeIndex],
								EnergyCounter_t:=GlobalEnergyCounter_t[GeoNodeIndex],KeyQty:=2);
				(*aggiorno controllo stato dei nodi *)
				LuxGeolumenNodes[GeoNodeIndex].checkStatusANDPresence();
				LuxGeolumenNodesAlignFlags[GeoNodeIndex]:=isGeolumenEqualStatus(LuxGeolumenNodes[GeoNodeIndex].desideredState, LuxGeolumenNodes[GeoNodeIndex].feedbackState);
				LuxGeolumenNodesCurrent[GeoNodeIndex]:=LuxGeolumenNodes[GeoNodeIndex].feedbackState.LampCurrent;
			END_IF
		END_FOR

		(*gestione dei log con temporizzazione *)
		maxLoggerRow:=MAX_LUXNUM/10 + SEL((MAx_LUXNUM MOD 10) =0,1,0);

		(*log periodico, 'logtrig' *)
		IF SyncLogRequest = FALSE THEN

			timingLuxBase:=TIME_LUX_LOG_NORMAL;
			timingAstroBase:=TIME_ASTRO_LOG_NORMAL;

			FOR tIndex:=1 TO maxLoggerRow DO
				TimerLogLux[tIndex](IN:=NOT TimerLogLux[tIndex].Q,PT:=timingLuxBase+INT_TO_TIME(TIME_TO_INT(t#5s)*tIndex));
					IF TimerLogLux[tIndex].Q THEN
						(* Trig logger *)
						objLuxLog(tIndex);
					END_IF
			END_FOR

			FOR tIndex:=1 TO maxLoggerRow DO
				TimerLogAstro[tIndex](IN:=NOT TimerLogAstro[tIndex].Q,PT:=timingAstroBase+INT_TO_TIME(TIME_TO_INT(t#5s)*tIndex));
				IF TimerLogAstro[tIndex].Q THEN
					(* Trig logger *)
					objAstroLog(tIndex);
				END_IF
			END_FOR

		(* log su richiesta *)
		ELSE

			IF logRowLux < maxLoggerRow THEN
				FOR tIndex:=1 TO maxLoggerRow DO
					TimerLogLuxSync[tIndex](IN:=NOT TimerLogLuxSync[tIndex].Q,PT:=timingLuxBase+INT_TO_TIME(TIME_TO_INT(t#5s)*tIndex));
					IF TimerLogLuxSync[tIndex].Q AND TimerLogLuxSyncDone[tIndex] = FALSE THEN
						(* Trig logger *)
						objLuxLog(tIndex);
						logRowLux:=(logRowLux+1) MOD (maxLoggerRow+1) + logRowLux/(maxLoggerRow+1);
						TimerLogLuxSyncDone[tIndex]:=TRUE;
					END_IF
				END_FOR
			END_IF

			IF logRowAstro < maxLoggerRow THEN
				FOR tIndex:=1 TO maxLoggerRow DO
					TimerLogAstroSync[tIndex](IN:=NOT TimerLogAstroSync[tIndex].Q,PT:=timingAstroBase+INT_TO_TIME(TIME_TO_INT(t#5s)*tIndex));
					IF TimerLogAstroSync[tIndex].Q AND TimerLogAstroSyncDone[tIndex] = FALSE THEN
						(* Trig logger *)
						objAstroLog(tIndex);
						logRowAstro:=(logRowAstro+1) MOD (maxLoggerRow+1) + logRowLux/(maxLoggerRow+1);
						TimerLogAstroSyncDone[tIndex] :=TRUE;
					END_IF
				END_FOR
			END_IF

			IF logRowAstro>=maxLoggerRow AND logRowLux>=maxLoggerRow THEN SyncLogRequest:=FALSE; END_IF

		END_IF


	(* stato S_RELOAD
	     - ricarica su richiesta il file associato
	*)
	S_RELOAD:

		(*ricaricamento file di configurazione: azzero tutti i Lux, Astr GeolumenNodes e ricomincio da capo *)
		LogEv(EL_Wrn,EO_SYS,0,1,CONCAT('System_reload_config_file',WORD_TO_STRING(Plant_SW_VER)));
		FOR counter := 1 TO MAX_LUXNUM DO
			TabListLux[counter].LuxID_Geolumen:=0;
			TabListLux[counter].MacAdd:=0;
			TabListLux[counter].MacAddH:=0;
			TabListLux[counter].MacAddL:=0;
			TabListLux[counter].StMacAdd:='';
			TabListLux[counter].LuxNumber:=0;
			TabListLux[counter].xCoupled:=FALSE;
			LuxElement[counter].ID:=0;
			ASTR[counter].ID:=0;
			LuxGeolumenNodes[counter].ID_Lux:=0;
			LuxGeolumenNodes[counter].ID_Geolumen:=0;
		END_FOR
		FOR counter := 0 TO MAX_ARRAY_MSG  DO
				MsgRecBuffer[i].Msg:='';
				MsgRecBuffer[i].MsgType := COMPLETED;
				MsgRecBuffer[i].dwMacAdd:=0;
		END_FOR

		Sys.Status:=S_STARTUP;

(* altrimenti vado in S_STARTUP *)
ELSE
	Sys.Status:=S_STARTUP;
END_CASE;
END_ACTION

(* POU ClevergyUtils/TCP_Logger/Logger_Proc, ST *)
PROGRAM Logger_Proc
VAR
	c1:         	TCPCLIENT;

	Open:	    	BOOL;
	IpAddr:			DWORD;
	InetAddr:		DWORD;
	Connected:  	BOOL;
	Error:      	DINT;
	TxTrig:     	BOOL;
	RxData:			ARRAY [0..MAX_RECEIVE_TCP_CLIENT] OF BYTE;
	RxLen:			DINT;

	Retry:			BYTE;	(* Counter for connection retries *)
	Recovered:		BYTE;	(* Counter for recovered unsent messages *)

	i:				DINT;
	pos:			DWORD;
	hFile:			DWORD;

END_VAR
(*=== State machine ===*)
CASE Logger.Status OF

	S_Logger_UNKNOWN:
		(* Startup *)
		Logger.SendReq:=FALSE;
		Open:=FALSE;
		Logger.Status:=S_Logger_IDLE;

	S_Logger_IDLE:
		(* Wait request *)
		IF Logger.SendReq THEN
			(* Resolve server name or use static IP *)
			IF LEN(Logger_SERVER)=0 THEN
				InetAddr:=SysSockInetAddr(Logger_IP);
			ELSE
				IpAddr:=SysSockGetHostByName(ADR(Logger_SERVER));	(* Get the IP address by the DNS *)
				DWORDSWAP(pIn:=ADR(IpAddr), pOut:=ADR(InetAddr));
			END_IF
			TxTrig:=FALSE;
			RxLen:=0;
			(* Open connection *)
			Open:=TRUE;
			Logger.Status:=S_Logger_WAITCONN;
		END_IF

	S_Logger_WAITCONN:
		(* Wait connection *)
		IF Connected THEN
			(* Send data *)
			TxTrig:=TRUE;
			Logger.Status:=S_Logger_WAITTX;
		END_IF
		IF Error>0 THEN
			Open:=FALSE;
			Logger.Status:=S_Logger_ERROR;
		END_IF

	S_Logger_WAITTX:
		(* Wait transmission *)
		IF NOT TxTrig THEN
			Logger.Status:=S_Logger_WAITRESP;
		END_IF
		IF Error>0 THEN
			Open:=FALSE;
			Logger.Status:=S_Logger_ERROR;
		END_IF

	S_Logger_WAITRESP:
		(* Wait response *)
		IF Connected=FALSE (* OR TIMEOUT!! *) THEN
			Open:=FALSE;
			(* Check response *)
			IF RxLen>=4 AND CHKSTRING(pString:=ADR(RxData), pPattern:=ADR(Logger_CHECK)) THEN
			(* If "RxLen" is of the right size and function "CHKSTRING" has not return "FALSE"	*)
				Logger.SendReq:=FALSE;
				Retry:=0;
				(* Check unsent messages to flush *)
				IF Recovered<Logger_RecoverMsgs THEN
					MsgChk();
					IF Logger.SendReq=TRUE THEN
						Recovered:=Recovered+1;
					ELSE
						Recovered:=0;
					END_IF
				ELSE
					Recovered:=0;
				END_IF
				Logger.Status:=S_Logger_IDLE;
			ELSE
				Logger.Status:=S_Logger_ERROR;
			END_IF
		END_IF

	S_Logger_ERROR:
		(* Connection error or send failure *)
		Retry:=Retry+1;
		IF Retry>Logger_ConnRetries THEN
			(* Save message as unsent *)
			MsgSave();
			Logger.SendReq:=FALSE;
			Retry:=0;
		END_IF
		Logger.Status:=S_Logger_IDLE;

ELSE
	Logger.Status:=S_Logger_UNKNOWN;
END_CASE


(*=== Execute client lib ===*)
c1(
	xOpenConnection			:= Open,
	dwInetAddr 				:= InetAddr,
	wPortNumber				:= Logger_PORT,
	ptSendData				:= ADR(Logger.SendData),
	diSendCount				:= Logger.SendLen,
	tConnectWatchdogTime	:= t#10s,
	xStartSend				:= TxTrig,
	aReceiveBuffer			:= RxData,
	diReceiveCount			:= RxLen,
	xConnected				=> Connected,
	diError					=> Error
);

(*=== Process Rx data ===*)
(*IF RxLen>0 THEN
	RxLen:=0;
END_IF*)
END_PROGRAM
ACTION MsgChk:
(* Open index file *)
hFile:=SysFileOpen(Logger_IndexFile,'r');
IF hFile=0 THEN
	(* File doesn't exist, no pending message *)
	RETURN;
END_IF
(* Search oldest message to recover *)
SysFileSetPos(hFile,Logger.LastIdxPos);		(* Set the pointer to last position *)
Logger.SendLen:=0;
REPEAT
	SysFileRead(hFile, ADR(Logger.SendIdx), SIZEOF(Logger.SendIdx));
	pos:=SysFileGetPos(hFile);
	SysFileRead(hFile, ADR(Logger.SendLen), SIZEOF(Logger.SendLen));
UNTIL
	SysFileEOF(hFile) OR Logger.SendLen<>0		(* If equal to 0 means data not stored or deleted *)
END_REPEAT
SysFileClose(hFile);
(* Delete index file when all messages are recovered *)
IF Logger.SendLen=0 THEN
	Logger.LastIdxPos:=0;
	SysFileDelete(Logger_IndexFile);
	RETURN;
END_IF
(* Recover message data *)
hFile:=SysFileOpen(Logger_DataFile,'r');
IF hFile<>0 THEN
	SysFileSetPos(hFile,Logger.SendIdx);
	SysFileRead(hFile,ADR(Logger.SendData),Logger.SendLen);
	Logger.SendReq:=TRUE;									(* Re-trigger another transmission *)
	SysFileClose(hFile);
END_IF
(* Clear index entry *)
hFile:=SysFileOpen(Logger_IndexFile,'rw'); (*diego: change from 'a' *)
IF hFile<>0 THEN
	SysFileSetPos(hFile,pos);
	i:=0;
	SysFileWrite(hFile, ADR(i), 4);			(* Since the size is in number of byte, that clears only the Idx, not the Len *)
	Logger.LastIdxPos:=SysFileGetPos(hFile);
	SysFileClose(hFile);
END_IF
END_ACTION
ACTION MsgSave:
(* Add log position in recovery indexes *)
hFile:=SysFileOpen(Logger_IndexFile,'a');
SysFileWrite(hFile, ADR(Logger.SendIdx), SIZEOF(Logger.SendIdx));
SysFileWrite(hFile, ADR(Logger.SendLen), SIZEOF(Logger.SendLen));
SysFileClose(hFile);
END_ACTION

(* POU ClevergyUtils/TCPCLIENT, ST *)
FUNCTION_BLOCK TCPCLIENT
(***********************************************************************************************************	*)
(* Version: 1.3b                        			          													*)
(* Date: 28.10.2014                   				          							            			*)
(***********************************************************************************************************	*)
(* WAGO Kontakttechnik GmbH Hansastr. 27 32423 Minden(Westf.)													*)
(* Tel. +0049 571/887-0 Fax. +0049 571/887-0																	*)
(* Author: VB																									*)
(***********************************************************************************************************	*)
(*Description:	A TCP client to read and write data with additional connection watchdog							*)
(*History:																										*)
(*Version 1.3b: 28.10.2014: Use DWORD address for IP (Andrea Ravasio)											*)
(*Version 1.3: 11.02.2011: Changes according to 750-880/881											 			*)
(*Version 1.2: 29.08.2007 Bugfix TCP Client																		*)
(*Version 1.1: 15.01.2007 Changes according to FW11																*)
(*Version 1.0: 09.03.2006 Release																				*)
(***********************************************************************************************************	*)
VAR CONSTANT
	STATE_CREATE     				 : BYTE:= 0;
	STATE_OPEN     					 : BYTE:= 1;
	STATE_IOCTL    					 : BYTE:= 2;
	STATE_CONNECT     				 : BYTE:= 10;
	STATE_TX       					 : BYTE:= 20;
	STATE_RX       					 : BYTE:= 30;
	STATE_CLOSE    					 : BYTE:= 40;
	STATE_ERROR_TRAP			     : BYTE:= 200;
END_VAR

VAR_INPUT
	xOpenConnection					: BOOL;
	dwInetAddr						: DWORD; (* <== Use SysSockInetAddr() value or
													swapped bytes order of SysSockGetHostByName() value *)
	wPortNumber						: WORD;
	ptSendData						: POINTER TO ARRAY[0..MAX_SEND_TCP_CLIENT] OF BYTE;
	diSendCount						: DINT;
	tConnectWatchdogTime		    : TIME := t#10s;
END_VAR
VAR_OUTPUT
	xConnected						: BOOL;
	diError 						: DINT := 0;
END_VAR
(* ErrorCodes -----------------------------------------
	16#8001 => No socket descriptor available 
	16#8002 => SysSockSend returns -1 
	16#8003 => Socket was "gracefully closed" 
	16#8004 => switching to none blocking mode fails
	16#8005 => SysSockClose() returns FALSE 
    16#8006 => SysSockConnect() fails
    16#8007 => SysSockSend() fails
	16#8008 => error state machine 
	16#8009 => timeout while waiting for data from server 
------------------------------------------------------------*)
VAR_IN_OUT
	xStartSend							: BOOL;
	aReceiveBuffer						: ARRAY [0..MAX_RECEIVE_TCP_CLIENT] OF BYTE;
	diReceiveCount						: DINT;
END_VAR
VAR
	m_State								: BYTE := 0;
	m_ReceiveBuffer						: ARRAY [0..MAX_RECEIVE_TCP_CLIENT_SOCKET] OF BYTE;
	m_Socket							: DINT;
	m_AddressInfo						: SOCKADDRESS;
	m_BytesReceived						: DINT;
	m_diReturn							: DINT;
	m_xReturn							: BOOL;
	m_IoCtlParameter  					: DINT := 1; (* IOCTL-Parameter for non-blocking mode of sockets *)
	i									: INT;
	T_Connect							: TON;
	m_count								: DINT;
	diOption							: DINT := 1;
	m_Blocking   						: DINT := 0;
END_VAR
IF xOpenConnection THEN
	(* State maschine *)
	CASE  m_State OF

	(* -------------------------------------------------------------------------*)
	STATE_CREATE:
			(* create socket descriptor*)
			m_Socket := SysSockCreate(diAddressFamily	:= SOCKET_AF_INET,
													 diType		:= SOCKET_STREAM,
													 diProtocol := SOCKET_IPPROTO_TCP);
			IF m_Socket >= 0 THEN
			(*Set Push-Bit*)
				IF ADR(%MW0)=16#30000000  OR ADR(%MW0)=16#20000000 THEN (*841 or 881*)
					SysSockSetOption(
						diSocket:=m_Socket,
						diLevel:=6,
						diOption:=SOCKET_TCP_NODELAY,
						pOptionValue:=ADR(diOption),
						diOptionLength:=SIZEOF(diOption));
				ELSE
						;
				END_IF
				m_State := STATE_IOCTL; (* succesful *)
			ELSE
				diError := 16#8001;  (* no socket descriptor available *)
				m_State := STATE_ERROR_TRAP;
			END_IF

	(* -------------------------------------------------------------------------*)
	STATE_IOCTL: (* change  socket mode  to none blocking *)
		m_diReturn := SysSockIoctl( m_Socket, SOCKET_FIONBIO, ADR(m_IoCtlParameter));
		IF m_diReturn <> 0 THEN
			m_AddressInfo.sin_family := SOCKET_AF_INET;
			m_AddressInfo.sin_port := SysSockNtohs(wPortNumber);
			m_AddressInfo.sin_addr := dwInetAddr;
			m_State := STATE_CONNECT;
		ELSE
			diError := 16#8004;  (* switching to none blocking mode fails *)
			m_State := STATE_ERROR_TRAP;
		END_IF


	(* -------------------------------------------------------------------------*)
	STATE_CONNECT: (* connect with server *)
		T_Connect(IN:=TRUE , PT:=tConnectWatchdogTime);(*activate watchdog for establishing connection to a server*)
		m_xReturn := SysSockConnect ( m_Socket, ADR(m_AddressInfo),  SIZEOF(m_AddressInfo));
		IF m_xReturn THEN (* succesful *)
			IF xStartSend THEN
				m_State := STATE_TX;(*transmit data*)
			ELSE
				m_State := STATE_RX;(*wait for data from server*)
			END_IF
			xConnected:=TRUE;
			T_Connect(IN:=FALSE);
		ELSE
			IF T_Connect.Q THEN
				diError := 16#8006;  (* connect fails *)
				xConnected:=FALSE;
				T_Connect(IN:=FALSE);
				m_State := STATE_ERROR_TRAP;
				SysSockClose( m_Socket);
			ELSE
				m_State := STATE_CONNECT;(*client still  tries to set up connection*)
			END_IF
		END_IF


	STATE_TX:	 (* send TCP-message *)
		m_diReturn := SysSockSend(diSocket := m_Socket,
								  pbyBuffer := ADR(ptSendData^[0]),
								  diBufferSize := diSendCount-m_count,
								  diFlags := 0);

		CASE m_diReturn OF
		-1:	(* ERROR *)
			T_Connect(IN:=TRUE , PT:=CONNECT_WATCHDOG_TIME);(*activate watchdog to check communication*)
			IF t_Connect.Q THEN
				diError := 16#8007;
				T_Connect(IN:=FALSE);
				m_State:=STATE_CLOSE;
			END_IF
		0: (* socket was "gracefully closed" *)
			m_State := STATE_CLOSE;
			diError := 16#8003;
		ELSE (* succesful *)
			m_count:=m_count+m_diReturn;
			IF m_count>=diSendCount THEN
				diError := 16#0000;
				m_State := STATE_RX;
				m_count:=0;
				xStartSend:=FALSE;
			END_IF
			T_Connect(IN:=FALSE);
		END_CASE

	(* -------------------------------------------------------------------------*)
	STATE_RX: (* process receive data *)
			m_BytesReceived := SysSockRecv(	diSocket 	:= m_Socket,
										pbyBuffer 	:= ADR(m_ReceiveBuffer),		(* Address of receive buffer *)
										diBufferSize:= SIZEOF(m_ReceiveBuffer),
										diFlags		:= 0);

			CASE m_BytesReceived OF
			-1:	(* No data available or error occured *)
				T_Connect(IN:=TRUE , PT:=tConnectWatchdogTime);(*activate watchdog to check communication*)
				IF t_Connect.Q THEN
					diError:=16#8009;
					T_Connect(IN:=FALSE);
					m_State:=STATE_CLOSE;
				END_IF
				IF xStartSend THEN
					m_State:=STATE_TX	;(* WAIT IN THIS STATE  and check for arriving data or new send command*)
				END_IF;
			0: (* socket was "gracefully closed"  *)
				m_State:=STATE_CLOSE;
				diError := 16#8003;
			ELSE (* succesful *)
				diError := 16#0000;
				T_Connect(IN:=FALSE);
				(* Copy received data into receive buffer *)
				FOR i:= 0 TO DINT_TO_INT(m_BytesReceived	)-1 DO
					aReceiveBuffer[diReceiveCount]:= m_ReceiveBuffer[i];
					diReceiveCount:=(diReceiveCount+1) MOD SIZEOF(aReceiveBuffer);
				END_FOR

			END_CASE

	(* -------------------------------------------------------------------------*)
	STATE_CLOSE : (* close socket *)
		IF ADR(%MW0)=16#30000000  OR ADR(%MW0)=16#20000000 THEN (*841 or 881*)
			;
		ELSE
			SysSockShutdown(m_Socket, 0);;(*870*)
		END_IF
		m_xReturn := SysSockClose( m_Socket);
		m_Socket := -1;
		m_State := 0; (* succesful *)
		xConnected:=FALSE;
		T_Connect(IN:=FALSE);
	(* -------------------------------------------------------------------------*)
	STATE_ERROR_TRAP: (* error handling *)
		xConnected:=FALSE;

	ELSE  (* Bad FSM code trap  *)
			m_State:= STATE_ERROR_TRAP;
			diError:= 16#8008;
	END_CASE

ELSE(*close connection*)
	IF m_Socket >= 0 THEN
		IF ADR(%MW0)=16#30000000  OR ADR(%MW0)=16#20000000 THEN (*841 or 881*)
			;
		ELSE
			SysSockShutdown(m_Socket, 0);;(*870*)
		END_IF
		SysSockClose( m_Socket);
	END_IF
	m_Socket := -1;
	diError := 16#0000;
	m_State := STATE_CREATE;
	xConnected:=FALSE;
	T_Connect(IN:=FALSE);
END_IF
END_FUNCTION_BLOCK

(* POU ClevergyUtils/DWORDSWAP, ST *)
FUNCTION DWORDSWAP:BOOL
VAR_INPUT
	pIn:POINTER TO ARRAY[1..4] OF BYTE;
	pOut:POINTER TO ARRAY[1..4] OF BYTE;
END_VAR
VAR
END_VAR
pOut^[1]:=pIn^[4];
pOut^[2]:=pIn^[3];
pOut^[3]:=pIn^[2];
pOut^[4]:=pIn^[1];
END_FUNCTION

(* POU ClevergyUtils/CHKSTRING, ST *)
FUNCTION CHKSTRING : BOOL
VAR_INPUT
	pString: POINTER TO BYTE;
	pPattern: POINTER TO BYTE;
END_VAR
VAR
END_VAR
CHKSTRING:=TRUE;
WHILE pPattern^<>0 AND CHKSTRING DO
	IF pPattern^<>pString^ THEN CHKSTRING:=FALSE; END_IF
	pString:=pString+1;
	pPattern:=pPattern+1;
END_WHILE
END_FUNCTION

(* POU TCP_Remote/Remote_Proc, ST *)
PROGRAM Remote_Proc
VAR
	s1:         	TCPSERVER;
	Enable: 		BOOL;
	Connected: 		BOOL;
	Error: 			DINT;

	TxData:			ARRAY [0..MAX_SEND_TCP_SERVER] OF BYTE;
	TxLen:			DINT;
	TxTrig:			BOOL;

	RxData:			ARRAY [0..MAX_RECEIVE_TCP_SERVER] OF BYTE;
	RxLen:			DINT;

	Status:			DINT;

	(* Command interpreter *)

	Cmd_Buf:		ARRAY [0..MAX_RECEIVE_TCP_SERVER] OF BYTE;
	Cmd_Buf_U16:	POINTER TO WORD;
	Cmd_Buf_INT:	POINTER TO INT;
	Cmd_BufLen:		WORD;
	Cmd_St:			WORD;

	Cmd_Obj:		WORD;
	Cmd_ObjIdx:		WORD;
	Cmd_ObjIdx_Low:		BYTE;
	Cmd_ObjIdx_High:		BYTE;
	Cmd_C:			WORD;
	Cmd_R:			WORD;
	Cmd_CLen:		WORD;
	Cmd_RLen:		WORD;

	i : WORD;
	j : INT;
	s2 : STRING;

	(* per aggiornare la data e l'ora *)
	SetAnno: INT;
	SetMese: INT;
	SetGiorno: INT;
	SetOra: INT;
	SetMinuti: INT;
	SetSecondi: INT;

	Plant_SW_VER: BOOL;
        	 (* specific for lux *)
	x: INT;
	NewValueTimer : DWORD;
	ModeFromPlc:EN_Modality;

	obj_ASTR_aux:obj_ASTR_aux;

END_VAR
(*=== State machine ===*)
CASE Status OF
	0: (* Startup *)
		TxLen:=0; TxTrig:=FALSE;
		RxLen:=0;
		Enable:=TRUE;
		Status:=1;

	1: (* Wait incoming connection *)
		IF Connected THEN
			(* Log access *)(*
			LogEv(EL_Log,EO_VPN,1,5,'Remote');*)
			(* Send welcome message *)(*
			ADDSTRING(pTxData:=ADR(TxData), pString:=ADR(Remote_WELCOME), TxLen:=TxLen);
			TxTrig:=TRUE;*)
			(* Reset vars *)
			Cmd_BufLen:=0;
			Cmd_St:=0;
			Status:=2;
		END_IF
		IF Error>1 THEN
			Enable:=FALSE;
			Status:=0;
		END_IF

	2: (* Wait command *)
		IF RxLen>0 THEN
			(*=== Interpreter start ===*)
			IF Cmd_BufLen+(RxLen/2)>=MAX_RECEIVE_TCP_SERVER THEN
				(* ERROR *)
				Cmd_BufLen:=0;
			ELSE
				i:=HEXTORAW(pString:=ADR(RxData), StringLen:=DINT_TO_WORD(RxLen), pData:=ADR(Cmd_Buf[Cmd_BufLen]));
				Cmd_BufLen:=Cmd_BufLen+i;
			END_IF
			IF Cmd_BufLen>=8 THEN
				Cmd_Buf_U16:=ADR(Cmd_Buf[6]);
				IF Cmd_BufLen>=(8+Cmd_Buf_U16^) THEN
					Cmd_CLen:=Cmd_Buf_U16^;
					Cmd_Buf_U16:=ADR(Cmd_Buf[0]); Cmd_Obj:=Cmd_Buf_U16^;
					Cmd_Buf_U16:=ADR(Cmd_Buf[2]); Cmd_ObjIdx:=Cmd_Buf_U16^;Cmd_ObjIdx_Low:=Cmd_Buf[2];Cmd_ObjIdx_High:=Cmd_Buf[3];
						(*fix per id maggiori di 255*)
						(*IF Cmd_Buf[3] <>0 THEN
							Cmd_ObjIdx:=ROL(Cmd_ObjIdx,8);
						END_IF*)
					Cmd_Buf_U16:=ADR(Cmd_Buf[4]); Cmd_C:=Cmd_Buf_U16^;
					(* Log command *)(*
					s2:='RCmd_';		s2:=CONCAT(s2,WORD_TO_STRING(Cmd_Obj));
					s2:=CONCAT(s2,'_'); s2:=CONCAT(s2,WORD_TO_STRING(Cmd_ObjIdx));
					s2:=CONCAT(s2,'_'); s2:=CONCAT(s2,WORD_TO_STRING(Cmd_C));
					s2:=CONCAT(s2,'_');	s2:=CONCAT(s2,WORD_TO_STRING(Cmd_CLen));
					LogEv(EL_Log,EO_VPN,1,6,s2);*)
					(* Execute command *)
					Command();
					Cmd_BufLen:=0;
				END_IF
			END_IF
			(*=== Interpreter end ===*)
			RxLen:=0;
		END_IF
		IF NOT Connected THEN
			Status:=0;
		END_IF

ELSE
	Status:=0;
END_CASE


(*=== Execute server lib ===*)
s1(
	xEnable				:= Enable,
	wPortNumber			:= Remote_PORT,
	tServerTimeOut		:= t#15m,
	ptSendData			:= ADR(TxData),
	diSendCount			:= TxLen,
	xStartSend			:= TxTrig,
	aReceiveBuffer		:= RxData,
	diReceiveCount		:= RxLen,
	xClientConnected	=> Connected,
	diError				=> Error
);
END_PROGRAM
ACTION Cmd_ASTR:
(* Check index *)
IF Cmd_ObjIdx < 1 THEN
	Cmd_R := 2; (* //id del lux fuori range*)
	RETURN ;
END_IF

x := 1 ;
WHILE ( x <=MAX_LUXNUM ) AND ( Cmd_ObjIdx <>  ASTR[ x ] . ID )  DO
	x := x + 1 ;
END_WHILE

(*
	Cmd_ObjIdx => logical id for Clevergy
	x=> where the object of ID Cmd_ObjIdx is placed inside the internal array
*)
IF  x <=MAX_LUXNUM AND Cmd_ObjIdx =  ASTR [ x ] . ID THEN

(* Process command *)
CASE Cmd_C OF

	1: (* GET PROFILE *)
		IF Cmd_CLen<>3 THEN
			Cmd_R:=4;
		ELSE
			(* Load profile *)
			CronEd.CN_Sel:=Cmd_ObjIdx;
			Cmd_Buf_U16:=ADR(Cmd_Buf[8]);
			CronEd.CN_YSel:=Cmd_Buf_U16^;
			CronEd.PR_Sel:=Cmd_Buf[10];
			CronEd.PR_Load_Exe();
			(* Copy data *)
			Cmd_RLen:=192;
			TxLen:=TxLen+RAWTOHEX(ADR(CronEd.PR.Setpoint),192,ADR(TxData[TxLen]));

		END_IF

	2: (* SET PROFILE *)
		IF Cmd_CLen<>(3+192) THEN
			Cmd_R:=4;
		ELSE
			(* Save profile *)
			CronEd.CN_Sel:=Cmd_ObjIdx;
			Cmd_Buf_U16:=ADR(Cmd_Buf[8]);
			CronEd.CN_YSel:=Cmd_Buf_U16^;
			CronEd.PR_Sel:=Cmd_Buf[10];
			MEMCPY(ADR(Cmd_Buf[11]),ADR(CronEd.PR.Setpoint),192);
			CronEd.PR_Save_Exe();

			ASTR[x].restartInternalCrono();
		END_IF

	5: (* GET CALENDAR MONTH *)
		IF Cmd_CLen<>3 THEN
			Cmd_R:=4;
		ELSE
			(* Load calendar *)
			CronEd.CN_Sel:=Cmd_ObjIdx;
			Cmd_Buf_U16:=ADR(Cmd_Buf[8]);
			CronEd.CN_YSel:=Cmd_Buf_U16^;
			CronEd.CA_Sel:=Cmd_Buf[10];
			CronEd.CA_Load_Exe();
			(* Copy data *)
			Cmd_RLen:=32;
			TxLen:=TxLen+RAWTOHEX(ADR(CronEd.CA.Profile),32,ADR(TxData[TxLen]));
		END_IF

	6: (* SET CALENDAR MONTH *)
		IF Cmd_CLen<>(3+32) THEN
			Cmd_R:=4;
		ELSE
			(* Save calendar *)
			CronEd.CN_Sel:=Cmd_ObjIdx;
			Cmd_Buf_U16:=ADR(Cmd_Buf[8]);
			CronEd.CN_YSel:=Cmd_Buf_U16^;
			CronEd.CA_Sel:=Cmd_Buf[10];
			MEMCPY(ADR(Cmd_Buf[11]),ADR(CronEd.CA.Profile),32);
			CronEd.CA_Save_Exe();
		END_IF

	9: (* CRON RESTART *)
		ASTR[x].restartInternalCrono();

	10: (* GET ASTR PARAMETERS *)


		Cmd_RLen:=10;
		TxLen:=TxLen + RAWTOHEX_BYTE(ADR(TxData[TxLen]),ASTR[x].preSunrise);
		TxLen:=TxLen + RAWTOHEX_BYTE(ADR(TxData[TxLen]),ASTR[x].postSunrise);
		TxLen:=TxLen + RAWTOHEX_BYTE(ADR(TxData[TxLen]),ASTR[x].preSunset);
		TxLen:=TxLen + RAWTOHEX_BYTE(ADR(TxData[TxLen]),ASTR[x].postSunset);
		TxLen:=TxLen + RAWTOHEX_BYTE(ADR(TxData[TxLen]),ASTR[x].twilightEveningMode);
		TxLen:=TxLen + RAWTOHEX_BYTE(ADR(TxData[TxLen]),ASTR[x].twilightMorningMode);



	11: (* SET ASTR PARAMETERS *)
		IF Cmd_CLen<>(12/2) THEN
			Cmd_R:=4;
		ELSE

			ASTR[x].preSunrise:=Cmd_Buf[8];
			ASTR[x].postSunrise:=Cmd_Buf[9];
			ASTR[x].preSunset:=Cmd_Buf[10];
			ASTR[x].postSunset:=Cmd_Buf[11];
			ASTR[x].twilightEveningMode:=Cmd_Buf[12];
			ASTR[x].twilightMorningMode:=Cmd_Buf[13];


			ASTR_CONFIG[x].preSunrise:=ASTR[x].preSunrise;
			ASTR_CONFIG[x].postSunrise:=ASTR[x].postSunrise;
			ASTR_CONFIG[x].preSunset:=ASTR[x].preSunset;
			ASTR_CONFIG[x].postSunset:=ASTR[x].postSunset;
			ASTR_CONFIG[x].twilightEveningMode:=ASTR[x].twilightEveningMode;
			ASTR_CONFIG[x].twilightMorningMode:=ASTR[x].twilightMorningMode;
			USE_RETAIN:=TRUE;

		END_IF


	12: (* SET ASTR SIMPLIFIED SCHEDULING *)

		IF Cmd_CLen<>(6) THEN
			Cmd_R:=4;
		ELSE

			obj_ASTR_aux(ASTR_ID:=ASTR[x].ID,cronEd:=CronEd, PE:=Cmd_Buf[8], QR:=Cmd_Buf[9], TN1_H:=Cmd_Buf[10], TN1_M:=Cmd_Buf[11], TN2_H:=Cmd_Buf[12], TN2_M:=Cmd_Buf[13] );
			obj_ASTR_aux.setSimplifedScheduling();
			ASTR[x].restartInternalCrono();

			IF obj_ASTR_aux.lastExecutionCode<0 THEN
				Cmd_R:=5;
			END_IF

		END_IF

	13: (* RESET ASTR SCHEDULING *)

		obj_ASTR_aux(ASTR_ID:=ASTR[x].ID,cronEd:=CronEd);
		obj_ASTR_aux.resetScheduling();


ELSE
	Cmd_R:=3;
END_CASE

ELSE
	Cmd_R := 2 ; (*//id del lux non presente in lista*)
END_IF
END_ACTION
ACTION Cmd_LUX:
(* Check index *)
IF Cmd_ObjIdx < 1 THEN
	Cmd_R := 2; (* //id del lux fuori range*)
	RETURN ;
END_IF

x := 1 ;
WHILE ( x <=MAX_LUXNUM ) AND ( Cmd_ObjIdx <>  LuxElement [ x ] . ID )  DO
	x := x + 1 ;
END_WHILE

IF  x <=MAX_LUXNUM AND  Cmd_ObjIdx =  LuxElement [ x ] . ID THEN

	(* Process command *)
 	CASE Cmd_C OF

		0 : (* Restore default functioning mode *)
			LuxElement [ x ] . CTRL_MODE := LuxElement [ x ] . CTRL_MODE_backUp ;
			LuxElement [ x ] (     WORKINGTIME := GlobalWorkingTime [ x ] ,
							POWERONCYCLES :=
							GlobalPowerOnCycles [ x ] ,
							ENERGYCOUNTER := GlobalEnergyCounter [ x ] ,
							ENERGYCOUNTER_T :=
							GlobalEnergyCounter_t [ x ] ,
							CtrlExton := KEYON ) ;

		1 : (* Reset statistic counter *)
			LuxElement [ x ] . StatReset (  WORKINGTIME := GlobalWorkingTime [ x ] ,
									POWERONCYCLES := GlobalPowerOnCycles [ x ] ,
									ENERGYCOUNTER :=GlobalEnergyCounter [ x ] ,
									ENERGYCOUNTER_T:= GlobalEnergyCounter_t [ x ] ,
									CtrlExton :=KEYON ) ;

		2 , 3 : (* Switch On (command=2) or Off (command=3) lux *)
			CASE Cmd_C OF
				2 : (*switch a Manuale ON*)
					LuxElement [ x ] . CTRL_MODE := 1 ; (*// Set to manuale ON *)
					LuxElement [ x ].DimmingValForManual:=LuxElement [ x ].MAX_DIMM_VALUE;
					LuxElement [ x ] (     WORKINGTIME := GlobalWorkingTime [ x ] ,
									POWERONCYCLES:= GlobalPowerOnCycles [ x ] ,
									ENERGYCOUNTER :=GlobalEnergyCounter [ x ] ,
									ENERGYCOUNTER_T :=GlobalEnergyCounter_t [ x ] ,
									CtrlExton := KEYON ) ;

				3 : (*switch a Manuale OFF*)
					LuxElement [ x ] . CTRL_MODE := 0 ; (*// Set to manuale OFF *)
					LuxElement [ x ].DimmingValForManual:=0;
					LuxElement [ x ] (     WORKINGTIME := GlobalWorkingTime [ x ] ,
									POWERONCYCLES:= GlobalPowerOnCycles [ x ] ,
									ENERGYCOUNTER :=GlobalEnergyCounter [ x ] ,
									ENERGYCOUNTER_T :=GlobalEnergyCounter_t [ x ] ,
									CtrlExton := KEYON ) ;

			END_CASE

		4 : (* Modify timer value *)
			IF  LuxElement [ x ] . CTRL_Mode = 03 THEN
				(*la modifica ha senso per i lux a timer*)
				NewValueTimer := BYTE_TO_DWORD ( Cmd_Buf [ 8 ] ) ;
				NewValueTimer := SHL ( NewValueTimer , 8 ) ;	
				NewValueTimer := NewValueTimer + BYTE_TO_DWORD ( Cmd_Buf [ 9 ] ) ;
				NewValueTimer := SHL ( NewValueTimer , 8 ) ;
				NewValueTimer := NewValueTimer + BYTE_TO_DWORD ( Cmd_Buf [ 10 ] ) ;
				NewValueTimer := SHL ( NewValueTimer , 8 ) ;
				NewValueTimer := NewValueTimer + BYTE_TO_DWORD ( Cmd_Buf [ 11 ] ) ;
				(*TabLuxPsg [ x ] . TimerOn := DWORD_TO_TIME ( NewValueTimer *1000 ) ;*) (*REMOVE THIS LINE *)

				FOR x := 1 TO MAX_LUXNUM DO
					IF LuxElement [ x ] . ID = Cmd_ObjIdx THEN
						LuxElement [ x ] . LuxTimer := DWORD_TO_TIME (NewValueTimer * 1000 ) ; (*//set del nuovo valore del timer del lux*)
					END_IF
				END_FOR
			ELSE
				Cmd_R := 3 ; (*//Comando errato / non previsto*)
			END_IF


	5:	(* get working mode*)
		Cmd_RLen:=2;
		ModeFromPlc:=LuxElement[x].CTRL_MODE;
		TxLen:=TxLen+RAWTOHEX(ADR(ModeFromPlc),2,ADR(TxData[TxLen]));

	6: (* SET MANUAL DIMMLEVEL*)
		IF Cmd_CLen<>(1) THEN
			Cmd_R:=4;
		ELSE
				IF(Cmd_Buf[8]>0) THEN
					LuxElement [x] . CTRL_MODE := 1 ; (*// Set to manuale on con dimm*)
					LuxElement [x].DimmingValForManual:=Cmd_Buf[8];
				ELSE
					LuxElement [x] . CTRL_MODE := 0 ; (*// Set to manuale off*)
					LuxElement [x].DimmingValForManual:=0;
				END_IF
				LuxElement [x] (    WORKINGTIME := GlobalWorkingTime [x ] ,
				POWERONCYCLES:= GlobalPowerOnCycles [x] ,
				ENERGYCOUNTER :=GlobalEnergyCounter [x] ,
				ENERGYCOUNTER_T :=GlobalEnergyCounter_t [x ] ,
									CtrlExton := KEYON ) ;
		END_IF
		ELSE
			Cmd_R := 3 ; (*//Comando errato / non previsto*)
		END_CASE
ELSE
	Cmd_R := 2 ; (*//id del lux non presente in lista*)
END_IF
END_ACTION
ACTION Cmd_SYS:
(* Check index *)
IF Cmd_ObjIdx<>0 THEN
	Cmd_R:=2;
	RETURN;
END_IF

(* Process command *)
CASE Cmd_C OF

	0: (* ECHO *)
		IF Cmd_CLen<>0 THEN
			TxLen:=0;
		END_IF

	1: (* LOG REQUEST *)
		LogTrig();

	2: (* REARM *)
		Sys.Warning:=FALSE;
		Sys.Alarm:=FALSE;
		Sys.AlarmStop:=FALSE;

	3: (* GET INFO1 *)
		Cmd_RLen:=6;
		TxLen:=TxLen+RAWTOHEX(ADR(Plant_SN),4,ADR(TxData[TxLen]));
		TxLen:=TxLen+RAWTOHEX(ADR(Plant_SW_VER),2,ADR(TxData[TxLen]));

	14: (*  Imposto data e ora del PLC  *)


			Cmd_Buf_U16:=ADR(Cmd_Buf[8]);
			SetAnno:= Cmd_Buf_U16^; 												(* Anno *)
			Cmd_Buf_U16:=ADR(Cmd_Buf[10]);
			SetMese:= Cmd_Buf_U16^;												 	(* mese *)
			Cmd_Buf_U16:=ADR(Cmd_Buf[12]);
			SetGiorno:=( Cmd_Buf_U16^);											 	(* Giorno *)
			Cmd_Buf_U16:=ADR(Cmd_Buf[14]);
			SetOra:=( Cmd_Buf_U16^); 												(* ora *)
			Cmd_Buf_U16:=ADR(Cmd_Buf[16]);
			SetMinuti:= ( Cmd_Buf_U16^);										 	(* Minuti *)
			Cmd_Buf_U16:=ADR(Cmd_Buf[18]);
			SetSecondi:= ( Cmd_Buf_U16^);										 	(* secondi *)

			SysRtcSetTime((SetDataTime(SetAnno,SetMese,SetGiorno,SetOra,SetMinuti,SetSecondi)));

ELSE
	Cmd_R:=3;
END_CASE
END_ACTION
ACTION Command:
(* Default response OK/NODATA *)
Cmd_R:=0;
Cmd_RLen:=0;
TxLen:=16;

(* Check object *)
CASE Cmd_Obj OF

	EO_SYS:
		Cmd_SYS();

	EO_LUX:
		Cmd_LUX();

	EO_ASTR:
		Cmd_ASTR();

ELSE
	Cmd_R:=3;
END_CASE

(* Generate response *)
IF TxLen>0 THEN
	RAWTOHEX(ADR(Cmd_Obj)	,2,ADR(TxData[ 0]));
	RAWTOHEX(ADR(Cmd_ObjIdx),2,ADR(TxData[ 4]));
	RAWTOHEX(ADR(Cmd_R)		,2,ADR(TxData[ 8]));
	RAWTOHEX(ADR(Cmd_RLen)	,2,ADR(TxData[12]));
	TxTrig:=TRUE;
END_IF
END_ACTION

(* POU ClevergyUtils/TCPSERVER, ST *)
FUNCTION_BLOCK TCPSERVER
(***********************************************************************************************************	*)
(* Version: 1.6                                    			          											*)
(* Date: 11.02.2011                                   					          							    *)
(***********************************************************************************************************	*)
(* WAGO Kontakttechnik GmbH Hansastr. 27 32423 Minden(Westf.)													*)
(* Tel. +0049 571/887-0 Fax. +0049 571/887-0																	*)
(* Author: VB																									*)
(***********************************************************************************************************	*)
(*Description:	A TCP server to read and write data													       		*)
(*Historie:																										*)
(*Version 1.6: 11.02.2011: Changes according to 750-880/881											 			*)
(*Version 1.5: 27.11.2008 Bugfix allow reuse port																*)
(*Version 1.4: 13.10.2008 Bugfix transmitting large data														*)
(*Version 1.3: 15.01.2007 Changes according to FW11																*)
(*Version 1.2: 09.03.2006 Changes for socket handle 0											       			*)
(*Version 1.1: 14.02.2005 Release																				*)
(***********************************************************************************************************	*)
VAR CONSTANT
	STATE_INIT     				 : BYTE:= 0;
	STATE_OPEN     				 : BYTE:= 1;
	STATE_TX       				 : BYTE:= 20;
	STATE_RX       				 : BYTE:= 30;
	STATE_CLOSE    				 : BYTE:= 40;
	STATE_ERROR_TRAP		 	 : BYTE:= 200;
END_VAR
VAR_INPUT
	xEnable    					: BOOL;	 (* Set TRUE to enable function block *)
	wPortNumber					: WORD;  (* Port *)
	tServerTimeOut				: TIME:=t#50s;
	ptSendData					: POINTER TO ARRAY[0..MAX_SEND_TCP_SERVER] OF BYTE;
	diSendCount					: DINT;
END_VAR
VAR_OUTPUT
	xClientConnected  			: BOOL:= FALSE;
	diError 					: DINT:= 0;
END_VAR
(* Status Codes -----------------------------------------
	16#8001 => No socket descriptor available 
	16#8002 => SysSockBind fails 
	16#8003 => SysSockListen fails 
	16#8004 => switching to none blocking mode fails
	16#8005 => SysSockClose() returns FALSE 
    16#8006 => SysSockConnect() fails
    16#8007 => SysSockSend() fails
	16#8008 => error state machine 
	16#8009 => timeout while waiting for data from server 
	16#0001 => server waiting for client to establish connection
------------------------------------------------------------*)
VAR_IN_OUT
	xStartSend					: BOOL;
	aReceiveBuffer				: ARRAY [0..MAX_RECEIVE_TCP_SERVER] OF BYTE;
	diReceiveCount				: DINT;
END_VAR

VAR
	m_State    					: BYTE:= 0;
	m_ReceiveBuffer				: ARRAY [0..MAX_RECEIVE_TCP_SERVER_SOCKET] OF BYTE;
	m_ServerSocket				: DINT:= SOCKET_INVALID;
	m_Socket					: DINT:= SOCKET_INVALID;
	m_AddressInfo				: SOCKADDRESS;
	m_BytesReceived				: DINT;
	m_diReturn					: DINT;
	m_xReturn					: BOOL;
	m_SizeSockadr				: DWORD;
	m_ConnectionWatchdog		: TON;
	m_Flags						: DINT;
	m_NoneBlocking   			: DINT:= 1;
	m_Blocking   				: DINT:= 0;
	i							: INT;
	m_count						: DINT;
	diOption					: DINT := 1;
	on: DINT;
END_VAR
IF xEnable THEN
	CASE m_State OF
		STATE_INIT:
			(* Create Socket *)
			m_ServerSocket:= SysSockCreate( SOCKET_AF_INET, SOCKET_STREAM, 0);
			IF m_ServerSocket = SOCKET_INVALID THEN
				(* *)
				diError:= 16#8001;
				m_State:= STATE_ERROR_TRAP;
				RETURN;
			ELSE
				;
			END_IF
			(* Address bindings *)
			(********************)
			on:=1;
			SysSockSetOption( m_ServerSocket, SOCKET_SOL, SOCKET_SO_REUSEADDR, ADR(on), SIZEOF(on) );

			m_AddressInfo.sin_family:= SOCKET_AF_INET;
			m_AddressInfo.sin_port  := SysSockHtons( wPortNumber);
			m_AddressInfo.sin_addr  := SOCKET_INADDR_ANY;
			IF NOT SysSockBind( m_ServerSocket, ADR(m_AddressInfo), SIZEOF(m_AddressInfo)) THEN
				diError:= 16#8002;
				m_State:= STATE_ERROR_TRAP;
				RETURN;
			END_IF
			(* Wait for connections *)
			(************************)
			IF NOT SysSockListen( m_ServerSocket, 1) THEN
				diError:= 16#8003;
				m_State:= STATE_ERROR_TRAP;
			END_IF

			(* Puts SOCKET in NonBlocking mode *)
			m_diReturn:= SysSockIoctl( m_ServerSocket, SOCKET_FIONBIO, ADR(m_NoneBlocking));

			m_State:= STATE_OPEN;


		STATE_OPEN: 	(* Waiting for incomming connection *)
				m_SizeSockadr:=SIZEOF(m_AddressInfo);
				m_Socket:= SysSockAccept( m_ServerSocket, ADR(m_AddressInfo), ADR(m_SizeSockadr));
				diError:=State_open;
				IF m_Socket <> SOCKET_INVALID THEN
					xClientConnected:=TRUE;
					(*Set Push-Bit:new V1.5*)
					IF ADR(%MW0)=16#30000000  OR ADR(%MW0)=16#20000000 THEN (*841 or 881*)
						SysSockSetOption(
							diSocket:=m_Socket,
							diLevel:=6,
							diOption:=SOCKET_TCP_NODELAY,
							pOptionValue:=ADR(diOption),
							diOptionLength:=SIZEOF(diOption));
					ELSE
							;
					END_IF
					SysSockIoctl( m_Socket, SOCKET_FIONBIO, ADR(m_NoneBlocking));
					m_State:= STATE_RX;
					diError:=0;
				END_IF

		STATE_RX:
					m_BytesReceived:= SysSockRecv( m_Socket, ADR(m_ReceiveBuffer), SIZEOF(m_ReceiveBuffer), 0);
					CASE m_BytesReceived OF
					-1:(*no data available or error occured*)
						m_ConnectionWatchdog(IN:=TRUE , PT:=tServerTimeOut );
						IF m_connectionWatchdog.Q THEN
							m_State:= STATE_CLOSE;
							m_ConnectionWatchdog(IN:=FALSE);(*reset connection watchdog*)
							diError := 16#8009;
						END_IF
					0:(* socket was "gracefully closed"  *)
						m_State:= STATE_CLOSE;
						diError := 16#8003;
					ELSE
						(* Copy received data into receive buffer *)
						(********************************)
						FOR i:= 0 TO DINT_TO_INT(m_BytesReceived	)-1 DO
							aReceiveBuffer[diReceiveCount]:= m_ReceiveBuffer[i];
							diReceiveCount:=(diReceiveCount+1) MOD SIZEOF(aReceiveBuffer);
						END_FOR

						m_ConnectionWatchdog(IN:=FALSE);(*reset connection watchdog*)
					END_CASE

				(*send data*)
				IF xStartSend	 THEN
					m_State := STATE_TX;
				END_IF

	STATE_TX:	 (* send TCP-message *)
		m_diReturn := SysSockSend(diSocket := m_Socket,
								  pbyBuffer := ADR(ptSendData^[m_count]),(*geändert V1.4 bisher: [0] *)
								  diBufferSize := diSendCount-m_count,
								  diFlags :=m_Flags);
		CASE m_diReturn OF
		-1:	(* ERROR or data could not yet be send (V1.3 due to new FW11) *)
			m_ConnectionWatchdog(IN:=TRUE , PT:=tServerTimeOut );
			IF m_connectionWatchdog.Q THEN
				m_State:= STATE_CLOSE;
				m_ConnectionWatchdog(IN:=FALSE);(*reset connection watchdog*)
				diError := 16#8007;
			END_IF
		0: (* socket was "gracefully closed"  *)
			m_State := STATE_CLOSE;
			diError := 16#8003;
		ELSE (* succesful *)
			m_count:=m_count+m_diReturn;
			IF m_count>=diSendCount THEN
				diError := 16#0000;
				m_State := STATE_RX;
				m_count:=0;
				xStartSend:=FALSE;
			END_IF
			m_ConnectionWatchdog(IN:=FALSE);(*reset connection watchdog*)
		END_CASE


		STATE_CLOSE:	(* Close the server *)

		IF ADR(%MW0)=16#30000000  OR ADR(%MW0)=16#20000000 THEN (*841 or 881*)
			;
		ELSE
			IF m_Socket>=0 THEN
				SysSockShutdown(m_Socket, 0);;(*870*)
			END_IF
		END_IF
		IF m_Socket>=0 THEN
			SysSockClose( m_Socket);
		END_IF
		xClientConnected:= FALSE;
		m_State:= STATE_OPEN; (* Try to open the server again *)
		m_ConnectionWatchdog(IN:=FALSE);(*reset connection watchdog*)

		STATE_ERROR_TRAP: (* Error Read/Write socket  *)
			m_State:= STATE_ERROR_TRAP;

	ELSE  (* Bad FSM code trap  *)
			m_State:= STATE_ERROR_TRAP;
			diError:= 16#8008;
	END_CASE;
ELSE
	IF m_State <> STATE_INIT THEN
		IF ADR(%MW0)=16#30000000  OR ADR(%MW0)=16#20000000 THEN (*841 or 881*)
			;
		ELSE
			IF m_Socket>=0 THEN
				SysSockShutdown(m_Socket, 0);;(*870*)
			END_IF
		END_IF
		IF m_Socket>=0 THEN
			SysSockClose( m_Socket);
		END_IF
		IF ADR(%MW0)=16#30000000  OR ADR(%MW0)=16#20000000 THEN (*841 or 881*)
			;
		ELSE
			IF m_ServerSocket>=0 THEN
				SysSockShutdown(m_ServerSocket, 0);;(*870*)
			END_IF
		END_IF
		IF m_ServerSocket>=0 THEN
			SysSockClose( m_ServerSocket);
		END_IF
		xClientConnected:= FALSE;
		diError:= 0;
		m_State:= STATE_init; (* Try to open the server again *)
		m_ConnectionWatchdog(IN:=FALSE);(*reset connection watchdog*)
	END_IF
END_IF
END_FUNCTION_BLOCK

(* POU obj_ASTR_aux, ST *)
FUNCTION_BLOCK obj_ASTR_aux
VAR_INPUT
	ASTR_ID:DWORD;
	PE: BYTE;
	QR:BYTE;
	TN1_H:BYTE;TN1_M:BYTE;
	TN2_H:BYTE;TN2_M:BYTE;
	cronEd:obj_CRON_EDITOR;
END_VAR
VAR_OUTPUT
	lastExecutionCommand:STRING(255);
	lastExecutionCode:INT;
END_VAR
VAR CONSTANT
	(*PROFILE TO BE USE FOR STOING THE SIMPLIFIED MODE VALUES *)
	SIMPLIFIED_MODE_PROFILE:BYTE:=10;
	DEFAULT_MODE_PROFILE:BYTE:=1;
	(*NUMBER OF THE LAST TIME SLOT => IS THE TOTAL NUMBER OF SLOTS -1*)
	LAST_TIME_SLOT_ID:BYTE:=95;
	LAST_CALENDAR_SLOT_ID:WORD:=384;
	ERROR_CODE_TN_NOT_INVALID:INT:=-1;
	ERROR_CODE_TN_NOT_COEHERENT:INT:=-2;
END_VAR
VAR
	tmp_Setpoint	: ARRAY [0..LAST_TIME_SLOT_ID] OF WORD;
	tmp_NightValue:WORD;
	slotTN1:WORD;
	slotTN2:WORD;
	i:INT;
	tmp_Profile : ARRAY[0..LAST_CALENDAR_SLOT_ID] OF BYTE;
END_VAR
;
END_FUNCTION_BLOCK
ACTION resetScheduling:
lastExecutionCommand:='resetScheduling';

FOR i:=0 TO LAST_CALENDAR_SLOT_ID DO
	tmp_Profile[i]:=DEFAULT_MODE_PROFILE;
END_FOR


FOR i:=1 TO 12 DO
	CronEd.CA_Sel:=INT_TO_BYTE(i);
	MEMCPY(ADR(tmp_Profile),ADR(CronEd.CA.Profile),32);
	CronEd.CA_Save_Exe();
END_FOR

lastExecutionCode:=0;
END_ACTION
ACTION setSimplifedScheduling:
lastExecutionCommand:='setSimplifiedScheduling';

(*check if times are valid)  *)
IF (TN1_H>23 OR TN2_H>23 OR TN1_M>59 OR TN2_M>59) THEN
	lastExecutionCode:=ERROR_CODE_TN_NOT_INVALID;
	RETURN;
END_IF


(*computing slot id for TN1 and TN2*)
slotTN1:=TN1_H*4+TN1_M/15;
slotTN2:=TN2_H*4+TN2_M/15;

(*check if times are coherent, must be slotTN2<> slotTN1
	exception: TN1 an TN2 zero
*)
IF (slotTN2<> 0 AND slotTN1<>0 AND NOT(slotTN2<>slotTN1) ) THEN
	lastExecutionCode:=ERROR_CODE_TN_NOT_COEHERENT;
	RETURN;
END_IF

(*computing setpoint*)

(*set all the slots to PE*)
FOR i:=0 TO LAST_TIME_SLOT_ID DO
	tmp_SetPoint[I]:=PE*10; (* 100 => 1000 *)
END_FOR

IF (slotTN2<> 0 AND slotTN1<>0 ) THEN

	(*computing night value as PE*QR% *)
	tmp_NightValue:=REAL_TO_WORD(BYTE_TO_WORD(PE)*10*(1-(BYTE_TO_REAL(QR)/100)));(* 100 => 1000 *)

	(* if TN2 < NT1 => external intervals *)
	IF(slotTN2<slotTN1) THEN

		(*assigning night value to the slot within TN1 and TN2*)

		FOR i:=0 TO slotTN2-1 DO
			tmp_SetPoint[i]:=tmp_NightValue;
		END_FOR


		FOR i:=slotTN1 TO LAST_TIME_SLOT_ID DO
			tmp_SetPoint[i]:=tmp_NightValue;
		END_FOR

	(* if TN2 < NT1 => internal intervals *)
	ELSIF (slotTN2>slotTN1) THEN

		FOR i:=slotTN1 TO slotTN2-1 DO
			tmp_SetPoint[i]:=tmp_NightValue;
		END_FOR

	END_IF

END_IF


CronEd.CN_Sel:=ASTR_ID;
CronEd.CN_YSel:=SYS.Time_Year;
CronEd.PR_Sel:=SIMPLIFIED_MODE_PROFILE;
MEMCPY(ADR(tmp_SetPoint),ADR(CronEd.PR.Setpoint),192);
CronEd.PR_Save_Exe();

FOR i:=0 TO LAST_CALENDAR_SLOT_ID DO
	tmp_Profile[i]:=SIMPLIFIED_MODE_PROFILE;
END_FOR


FOR i:=1 TO 12 DO
	CronEd.CA_Sel:=INT_TO_BYTE(i);
	MEMCPY(ADR(tmp_Profile),ADR(CronEd.CA.Profile),32);
	CronEd.CA_Save_Exe();
END_FOR

lastExecutionCode:=0;
END_ACTION

(* POU Plant_Objects/obj_CRON_EDITOR, ST *)
FUNCTION_BLOCK obj_CRON_EDITOR
(* === EDITOR CRONOGRAFO ===
   v1.0[16/04/15] - Versioning
   v1.1[19/05/15] - Create empty profile when not found
*)
VAR_INPUT

	CRONO_TYPE : STRING:='CR';

	(* Common selections *)
	CN_Sel:			DWORD:=1;
	CN_Act:			DWORD;
	CN_YSel:		WORD:=2015;
	CN_YAct:		WORD;

	(* Profile editor *)
	PR_Sel: 		BYTE:=1;
	PR_Act:			BYTE;
	PR_TT:			REAL;
	PR:				typ_Cron_Profile;
	(* Profile signals *)
	PR_Load:		BOOL;
	PR_Save:		BOOL;

	(* Calendar editor *)
	CA_Sel:			BYTE:=1; (* Calendar month selected *)
	CA_Act:			BYTE;    (* Calendar month active *)
	CA_DayF:		BYTE:=0;
	CA_DayL:		BYTE:=31;
	CA_TPR:			BYTE;
	CA:				typ_Cron_Calendar; (* Only used for first 32 entries *)
	(* Calendar signals *)
	CA_Load:		BOOL;
	CA_Save:		BOOL;

	(* Jolly editor *)
	JL:				ARRAY[0..9] OF typ_Cron_Jolly;
	(* Jolly signals *)
	JL_Load:		BOOL;
	JL_Save:		BOOL;

END_VAR
VAR_OUTPUT
	Message		: STRING;
END_VAR
VAR
	sFileName	: STRING;
	sFileMode	: STRING;
	hFile		: DWORD;
	Buf			: ARRAY[0..512] OF BYTE; (* AVOID THIS!! *)

	i			: WORD;
	ver			: BYTE;
	r1			: BOOL;
	r2			: DWORD;

END_VAR
IF PR_Load THEN PR_Load_Exe(); PR_Load:=FALSE; END_IF
IF PR_Save THEN PR_Save_Exe(); PR_Save:=FALSE; END_IF
IF CA_Load THEN CA_Load_Exe(); CA_Load:=FALSE; END_IF
IF CA_Save THEN CA_Save_Exe(); CA_Save:=FALSE; END_IF
IF JL_Load THEN JL_Load_Exe(); JL_Load:=FALSE; END_IF
IF JL_Save THEN JL_Save_Exe(); JL_Save:=FALSE; END_IF
END_FUNCTION_BLOCK
ACTION CA_Load_Exe:
sFileMode:='r';
FileOpen();

IF hFile<>0 THEN

	(* Read calendar month *)
	FOR i := 0 TO 31 DO
		r1:=SysFileSetPos(File:=hFile, Pos:=(1024 + ((CA_Sel-1)*32 + i)*4));
		r2:=SysFileRead(File:=hFile, Buffer:=ADR(CA.Profile[i]), Size:=1);
	END_FOR

	(* Close file *)
	SysFileClose(File:=hFile);

	(* Validate data *)
	CA_Act :=CA_Sel;
	CN_Act :=CN_Sel;
	CN_YAct:=CN_YSel;

	Message:='Calendar load OK';

END_IF
END_ACTION
ACTION CA_Save_Exe:
sFileMode:='rw';
FileOpen();

IF hFile<>0 THEN

	(* Write calendar month *)
	FOR i := 0 TO 31 DO
		r1:=SysFileSetPos(File:=hFile, Pos:=(1024 + ((CA_Sel-1)*32 + i)*4));
		r2:=SysFileGetPos(hFile);
		r2:=SysFileWrite(File:=hFile, Buffer:=ADR(CA.Profile[i]), Size:=1);
	END_FOR

	(* Close file *)
	SysFileClose(File:=hFile);

	Message:='Calendar save OK';

END_IF
END_ACTION
ACTION FileOpen:
(* Create current filename 'yyyyCRnn.DAT' *)
sFileName:=CONCAT(FilesPath,WORD_TO_STRING(CN_YSel));
sFileName:=CONCAT(STR1:=sFileName, STR2:=CRONO_TYPE);
IF CN_Sel<10 THEN
sFileName:=CONCAT(STR1:=sFileName, STR2:='0');
END_IF
sFileName:=CONCAT(STR1:=sFileName, STR2:=DWORD_TO_STRING(CN_Sel));
sFileName:=CONCAT(STR1:=sFileName, STR2:='.DAT');

(* Check file version and size! *)
(* ... *)

(* Open data file *)
hFile:=SysFileOpen(FileName:=sFileName, Mode:='r');

(* File not found *)
IF hFile=0 THEN
	Message:='File not found - created empty file';
	(* Create empty file *)
	hFile:=SysFileOpen(FileName:=sFileName, Mode:='w');
	MEMCLR(pDestinationAddress:=ADR(Buf), BytesToClear:=SIZEOF(Buf));
	FOR i := 0 TO 10239 BY 512 DO
		SysFileWrite(File:=hFile, Buffer:=ADR(Buf), Size:=512);
	END_FOR
	Buf[0]:=1;
	SysFileSetPos(File:=hFile, Pos:=0);
	SysFileWrite(File:=hFile, Buffer:=ADR(Buf), Size:=1);
END_IF

(* Close file *)
SysFileClose(File:=hFile);

(* Open data file *)
hFile:=SysFileOpen(FileName:=sFileName, Mode:=sFileMode);
END_ACTION
ACTION JL_Load_Exe:
sFileMode:='r';
FileOpen();

IF hFile<>0 THEN

	(* Read jolly *)
	r1:=SysFileSetPos(File:=hFile, Pos:=512);
	r2:=SysFileRead(File:=hFile, Buffer:=ADR(JL), Size:=SIZEOF(JL));

	(* Close file *)
	SysFileClose(File:=hFile);

	(* Validate data *)
	CN_Act:=CN_Sel;
	CN_YAct:=CN_YSel;

	Message:='Jolly load OK';

END_IF
END_ACTION
ACTION JL_Save_Exe:
sFileMode:='rw';
FileOpen();

IF hFile<>0 THEN

	(* Write selected profile *)
	r1:=SysFileSetPos(File:=hFile, Pos:=512);
	r2:=SysFileWrite(File:=hFile, Buffer:=ADR(JL), Size:=SIZEOF(JL));

	(* Close file *)
	SysFileClose(File:=hFile);

	Message:='Jolly save OK';

END_IF
END_ACTION
ACTION PR_Load_Exe:
sFileMode:='r';
FileOpen();

IF hFile<>0 THEN

	(* Read selected profile *)
	r1:=SysFileSetPos(File:=hFile, Pos:=(3072 + 512*PR_Sel));
	r2:=SysFileRead(File:=hFile, Buffer:=ADR(PR), Size:=SIZEOF(PR));

	(* Close file *)
	SysFileClose(File:=hFile);

	(* Validate data *)
	PR_Act:=PR_Sel;
	CN_Act:=CN_Sel;
	CN_YAct:=CN_YSel;

	Message:='Profile load OK';

END_IF
END_ACTION
ACTION PR_Save_Exe:
sFileMode:='rw';
FileOpen();

IF hFile<>0 THEN

	(* Write selected profile *)
	r1:=SysFileSetPos(File:=hFile, Pos:=(3072 + 512*PR_Sel));
	r2:=SysFileWrite(File:=hFile, Buffer:=ADR(PR), Size:=SIZEOF(PR));

	(* Close file *)
	SysFileClose(File:=hFile);

	Message:='Profile save OK';

END_IF
END_ACTION

(* POU ClevergyUtils/HEXTORAW, ST *)
FUNCTION HEXTORAW : WORD
VAR_INPUT
	pString		: POINTER TO BYTE;
	StringLen	: WORD;
	pData		: POINTER TO BYTE;
END_VAR
VAR
	xl: WORD;
	xi: WORD;
	xr: BYTE;
END_VAR
(* Convert transmitted hexadecimal data, encoded as string, back to hexadecimal format (see ASCII vs Hex table) *)
xl:=0;
xi:=0;

WHILE xi<StringLen DO

	IF pString^>=97 AND pString^<=102 THEN		(* Lower case letter "a..f" *)
		xr := pString^ - 87;
	ELSIF pString^>=65 AND pString^<=70 THEN	(* Upper case letter "A..F" *)
		xr := pString^ - 55;
	ELSIF pString^>=48 AND pString^<=57 THEN	(* Digit "0..9" *)
		xr := pString^ - 48;
	ELSE
		xr := 16;
	END_IF

	IF xr<16 THEN
		IF (xi AND 1)=0 THEN					(* Enter this if when even index (last digit is 0) *)
			pData^ := xr * 16;
		ELSE
			pData^ := pData^ + xr;				(* Enter this else when odd index (last digit is 1) *)
			pData := pData + 1;
			xl := xl + 1;
		END_IF
	END_IF

	xi := xi + 1;
	pString := pString + 1;

END_WHILE

HEXTORAW:=xl;									(* Number of word *)

(* NB Byte are transmitted MSB first *)
END_FUNCTION

(* POU ClevergyUtils/RAWTOHEX, ST *)
FUNCTION RAWTOHEX : WORD
VAR_INPUT
	pData: POINTER TO BYTE;
	DataLen: WORD;
	pString: POINTER TO BYTE;
END_VAR
VAR
	xl: WORD;
END_VAR
xl:=0;

WHILE DataLen>0 DO

	pString^ := (pData^ / 16#10) + 48 + (((pData^ / 16#10)/10)*7);
	pString:=pString+1;
	pString^ := (pData^ AND 16#0F)  + 48 + (((pData^ AND 16#0F)/10)*7);
	pString:=pString+1;
	pData:=pData+1;
	DataLen:=DataLen-1;
	xl:=xl+2;

END_WHILE

(*pString^:=0;*)

RAWTOHEX:=xl;
END_FUNCTION

(* POU ClevergyUtils/RAWTOHEX_BYTE, ST *)
FUNCTION RAWTOHEX_BYTE : BYTE
VAR_INPUT
	pString: POINTER TO  BYTE;
	DATUM : BYTE;

END_VAR
VAR
	tmp:BYTE;
END_VAR
	pString^ := (WORD_TO_BYTE(DATUM) / 16#10) + 48 + (((WORD_TO_BYTE(DATUM) / 16#10)/10)*7);
	pString:=pString+1;
	pString^ := (DATUM AND 16#0F)  + 48 + (((DATUM AND 16#0F)/10)*7);

	RAWTOHEX_BYTE:=2;
END_FUNCTION

(* POU ClevergyUtils/SetDataTime, ST *)
FUNCTION SetDataTime : DT
VAR_INPUT
	year : INT;
	month : INT;
	day : INT;
	hour : INT;
	minute : INT;
	second : INT;
END_VAR

VAR
	count : INT;
END_VAR
(* Creazione variabiletipo DT per creare Orario da dare al PLC *)


IF month > 2 THEN
	count := (month - 1) * 30;
	IF month > 7 THEN count := count + SHR(month - 3,1); ELSE count := count + SHR(month - 4,1); END_IF;
	(* chech for leap year and add one day if true *)
	IF SHL(year,14) = 0 THEN count := count + 1; END_IF;
ELSE
	count := (month - 1) * 31;
END_IF;


SetDataTime := DWORD_TO_DT(DATE_TO_DWORD( DWORD_TO_DATE((INT_TO_DWORD(count + day - 1) + SHR(INT_TO_DWORD(year) * 1461 - 2878169, 2)) * 86400))
				+ INT_TO_DWORD(SECOND)
				+ INT_TO_DWORD(MINUTE) * 60
				+ INT_TO_DWORD(HOUR) * 3600);
END_FUNCTION

(* POU GeoLumenWrapping/obj_GeolumenCoordinator, ST *)
FUNCTION_BLOCK obj_GeolumenCoordinator
VAR CONSTANT
	getStatusAllFeedback:STRING(255):='NWK_DISCOVER$R';
	setGlobalON:STRING(255):='GLO_SET_LIGHT:1023,1023,1023,0,0$R';
	setGlobalOFF:STRING(255):='GLO_SET_LIGHT:0,0,0,0,0$R';
END_VAR
VAR_INPUT
	ReceiveBufferPtr : POINTER TO typRing_Buffer;
	MsgRecBufferPtr : POINTER TO ARRAY[0..MAX_ARRAY_MSG ] OF type_MsgReceive;
END_VAR
VAR_OUTPUT
	LastMessage: STRING(255) := '';
END_VAR
VAR
	TimerCmdAdd:TON;
	LastSuperatoTime:DT;
	superatoAvanzo2:STRING(255):='';
	stringaSerialeCaso2: STRING(255);	(*  *)
	stringaSerialeCaso3:STRING(255):='';
	superatoAvanzo3:STRING(255):='';
	tempStringaCaso2:STRING(255);
	tempStringaCaso3:STRING(255);
	appoggioCaso2:STRING(255);
	appoggioCaso3:STRING(255);
	appoggioPosFullPrefix:INT;
	appoggioPosPartPrefix:INT;
	caso2NonPotuto:INT:=0;
	caso3NonPotuto:INT:=0;
	TimerSend : TON;
	xOpenPort		: BOOL := TRUE;
	xInitPort			: BOOL;
	xSendActive	: BOOL;
	xStartSend		: BOOL;
	SendString : STRING(255):='';
	pReceiveStr 	: POINTER TO STRING(255);
	StringaDaSeriale 	: STRING(255):='';
	tempStringa : STRING(255) := '';
	ArrayPos		: BYTE;
	LenghtStr	: INT;
	TrimStr1, TrimStr2,TrimNMEAS,TrimNMEAS_Med	: STRING(10);
	contFrame : INT :=0;
	StringCmp1, StringCmp2	: DINT;
	i :INT :=0;
	tempEnd: INT;
	tempBegin: INT;
	tempBegin0: INT;
	InitCom: BOOL;
	temp 		: BYTE;
	temp2		: INT;
	MyString	: STRING(255);
	pString1, pString2	: POINTER TO STRING(255);
	superatoTEMPSTRINGA:STRING(255):='';
	superatoSTRINGADASERIALE:STRING(255):='';
	tmpIndex:INT;
	maxStringaDaSerialeLength:INT:=0;
	maxConcat:INT:=0;
	x	: WORD;
	MacStr	: STRING (8);
	StrToSend	:STRING(255);
	counter, index	: WORD;
	StrLoc			: BYTE;
	StrSaveMacAdd	: STRING;
	StrSaveID		: STRING;
	Str				: STRING;
END_VAR
VAR CONSTANT
	ID_NODE_PREFIX:STRING:='IDN';
	PW0_PREFIX:STRING:='PW0';
	PW1_PREFIX:STRING:='PW1';
	PW2_PREFIX:STRING:='PW2';
	LAMP_CURRENT_PREFIX:STRING:='IAC';
	LAMP_POWER_PREFIX:STRING:='PAT';
	LAMP_VOLTAGE_PREFIX:STRING:='VAC';
	LQI_PREFIX:STRING:='LQI';
	FIELD_SEPARATOR:STRING:=';';
	ECHO_SET_LIGHT_ID_NODE_PREFIX:ARRAY[1..2] OF STRING(255):='>NDE_SET_LIGHT=','Gateway:NDE_SET_LIGHT:';
	ECHO_SET_LIGHT_NODE_SEPARATOR:ARRAY[1..2] OF STRING(255):=',','=';
	SET_LIGHT_PW_SEPARATOR:STRING:=',';
	PAR_PREFIX:STRING:='PAR';
END_VAR
VAR_INPUT
	statusNodeMessage : STRING(255);
	echoNodeMessage : STRING(255);
END_VAR
VAR_OUTPUT
	idNode : WORD;
	echoset_idNode : WORD;
	state: TYPE_LuxGeolumenStatus;
	echoCommandState: TYPE_LuxGeolumenStatus;
END_VAR
VAR
	pwm0 : WORD;
	pwm1 : WORD;
	pwm2 : WORD;
	lampCurrent:DWORD;lampVoltage:DWORD;lampPower:DWORD;
	lqiLast, lqiAvg, lqiMax : WORD:=0; lqiMin:WORD:=1023;
	countMSG:DWORD:=0;sumLqi:DWORD:=0;
	idNodeStart:INT;
	partialStringNode, partialStringPW0,partialStringPW1,partialStringPW2,partialStringLampCurrent,partialStringLampVoltage,partialStringLampPower, partialStringLqi:STRING(255);
	posSeparator:WORD;
	idPw0Start:INT;
	idPw1Start:INT;
	idPw2Start:INT;
	idLampCurrentStart:INT;idLampPowerStart:INT;idLampVoltageStart:INT;
	idLqiStart:INT;
	echoset_partialStringNode, echoset_partialStringPW0,echoset_partialStringPW1,echoset_partialStringPW2:STRING(255);
	echoset_posSeparator:WORD;
	echoset_idNodeStart:INT;
	echoset_idPw0Start:INT;
	echoset_idPw1Start:INT;
	echoset_idPw2Start:INT;
	echoset_pwm0 : WORD;
	echoset_pwm1 : WORD;
	echoset_pwm2 : WORD;

	idParCurrentStart:INT;idParVoltageStart:INT;idParPowerStart:INT;
	partialStringPar:STRING(255);
	lastPar:STRING(255);

END_VAR
VAR
	StrMin			: STRING(4);
	StrHour			: STRING(4);
	StartingState	: en_StartingState;
END_VAR
doSerialTransfer(); (* lettura/scrittura da porta seriale *)
getAndParseMessage2(); (*verifica della ricezione di un messaggio completo e parsing *)
SendAuth(); (*invia messaggio di autorizzazione per chi ne ha bisogno *)
ReadID(); (*esegue associazione ID --> Mac Address e lo scrive nella struttura TabListLux *)

(*AllCoupled();*) (* verifica se tutti i Mac Address sono acciopiati con l'ID*) (*eliminato, per mantenere dinamicità*)
END_FUNCTION_BLOCK
ACTION AllCoupled:
counter :=1;
xCoupledAll:=FALSE;
WHILE (counter<=MAX_GEOLUMENNODES) DO
	IF TabListLux[counter].xCoupled = FALSE THEN
		RETURN;
	END_IF
	counter:=counter+1;
END_WHILE
IF counter = MAX_GEOLUMENNODES+1 THEN
	xCoupledAll:=TRUE;
END_IF
END_ACTION
ACTION blockNodeAutoAdd:
SendString := 'CMD_AUTHORISE=0$R';
SendDataQueue(pTxData:=ADR(SendString));
SendDataQueue.addMessage();
END_ACTION
ACTION doSerialTransfer:
(* timer invio messaggi al coordinatore *)
TimerSend(IN:=NOT TimerSend.Q,PT:=GEOLUMEN_SEND_TIME);

(* di default leggo e basta*)
xStartSend:=FALSE;
SendString:='';

(* se non è scattato il timer invio messaggi al coordinatore, leggo e basta *)
IF NOT TimerSend.Q THEN

	COM0(	utRECEIVE_BUFFER := ReceiveBufferPtr^,
				ptSEND_BUFFER	:= ADR(SendString),
				xINIT			:=  xInitPort,
		     		xOPEN_COM_PORT 	:= TRUE,
				iBYTES_TO_SEND	:= LEN(SendString)+1,
				xSTART_SEND		:= xStartSend );

ELSE

	(* se il timer è scattato E ci sono messaggi in coda, invio *)
	IF(SendDataQueue.toBeSent>0) THEN
		SendDataQueue.getMessage();
		SendString:=SendDataQueue.StrToSend;
		xStartSend:=TRUE;
	END_IF

	COM0(	utRECEIVE_BUFFER := ReceiveBufferPtr^,
				ptSEND_BUFFER	:= ADR(SendString),
				xINIT				:=  xInitPort,
		     		xOPEN_COM_PORT 	:= TRUE,
				iBYTES_TO_SEND	:= LEN(SendString)+1,
				xSTART_SEND		:= xStartSend );

END_IF
END_ACTION
ACTION GetAndParseMessage:
IF pReceiveStr = 0 THEN
	pReceiveStr := ADR(ReceiveBufferPtr^.Data);
END_IF;

IF (ReceiveBufferPtr^.Index > 0 ) THEN
	StringaDaSeriale :=  pReceiveStr^ ;
	IF LEN(StringaDaSeriale) > maxStringaDaSerialeLength THEN
		maxStringaDaSerialeLength:=LEN(StringaDaSeriale);
	END_IF
	IF(LEN(tempStringa)+LEN(StringaDaSeriale)<=255) THEN
		tempStringa :=CONCAT(tempStringa, StringaDaSeriale);
	ELSE
		LastSuperatoTime:=SYS.Time_CT_DT;
		superatoTEMPSTRINGA:=tempStringa;
		superatoSTRINGADASERIALE:=StringaDaSeriale;
		tempStringa:='';
		tempStringa :=CONCAT(tempStringa, StringaDaSeriale);
	END_IF

	IF LEN(tempStringa)+LEN(StringaDaSeriale)>maxConcat THEN
		maxConcat:=LEN(tempStringa)+LEN(StringaDaSeriale);
	END_IF

	tempBegin:=FIND(tempStringa,'$R$N');

	IF(tempBegin>0) THEN
		LastMessage:=LEFT(tempStringa,tempBegin-1);
		tempStringa:='';

		MsgRecBuffer[ArrayPos].Msg:=LastMessage;

		LenghtStr:= LEN(MsgRecBuffer[ArrayPos].Msg);
		TrimStr1:=MID(MsgRecBuffer[ArrayPos].Msg, 3, 1); (*Isolo la sottostringa iniziale -  '#!#' *)

		IF(SysStrCmp(TrimStr1, '#.#') = 0) THEN
			TrimStr1:=MID(MsgRecBuffer[ArrayPos].Msg, 7, 4); (*Isolo la sottostringa iniziale - REQAUTH*)
			TrimStr2:=MID(MsgRecBuffer[ArrayPos].Msg, 4, 32); (*Isolo la sottostringa finale - STS0*)

			IF (SysStrCmp(TrimStr1, 'REQAUTH') = 0 AND SysStrCmp(TrimStr2, 'STS0') = 0) THEN
				MsgRecBuffer[ArrayPos].MsgType := REQAUTH0;
				(*contSts0:=contSts0+1;*)
			(*ELSIF (SysStrCmp(TrimStr1, 'REQAUTH') = 0 AND SysStrCmp(TrimStr2, 'STS1') = 0) THEN
				contSts1:=contSts1+1;*)
			ELSE
				TrimNMEAS:=MID(MsgRecBuffer[ArrayPos].Msg, 6, 4); (* Isolo la sottostringa iniziale - NMEAS*)
				IF (SysStrCmp(TrimNMEAS, 'NMEAS;') = 0  AND   FIND(MsgRecBuffer[ArrayPos].Msg,  '#!#' ) > 0) THEN
					MsgRecBufferPtr^[ArrayPos].MsgType := DATAREC;
					(*identifco a quale nodo lux geolumen si riferisce *)
					parseNodeStatus(statusNodeMessage:=MsgRecBufferPtr^[ArrayPos].Msg);
					IF idNode>=1 AND idNode<=MAX_LUXNUM THEN
						tmpIndex:=getGeolumenNodeByGeolumenId (idNode);
						IF(tmpIndex>0 AND tmpIndex<=MAX_LUXNUM) THEN
							LuxGeolumenNodes[tmpIndex](feedbackState:=state); LuxGeolumenNodes[tmpIndex].updateFeedbackState();
						END_IF
					END_IF
				END_IF

				(*TrimNMEAS_Med:=MID(MsgRecBuffer[ArrayPos].Msg, 8, 4); (* Isolo la sottostringa iniziale - NMEAS*)
				IF (SysStrCmp(TrimNMEAS, 'NMEASMED') = 0  AND   FIND(MsgRecBuffer[ArrayPos].Msg,  '#!#' ) > 0) THEN
					MsgRecBufferPtr^[ArrayPos].MsgType := DATAREC;
					(*identifco a quale nodo lux geolumen si riferisce *)
					parseNodeStatus(statusNodeMessage:=MsgRecBufferPtr^[ArrayPos].Msg);
					IF idNode>=1 AND idNode<=MAX_LUXNUM THEN
						tmpIndex:=getGeolumenNodeByGeolumenId (idNode);
						IF(tmpIndex>0 AND tmpIndex<=MAX_LUXNUM) THEN
							LuxGeolumenNodes[tmpIndex](feedbackState:=state); LuxGeolumenNodes[tmpIndex].updateFeedbackState();
						END_IF
					END_IF
				END_IF*)
			END_IF

		(*ELSIF  FIND(MsgRecBufferPtr^[ArrayPos].Msg,  '>NDE_SET_LIGHT=' ) = 1 (* Isolo la sottostringa iniziale - > *) THEN
			MsgRecBufferPtr^[ArrayPos].MsgType := ECHO;
			parseNodeEcho(echoNodeMessage:=MsgRecBufferPtr^[ArrayPos].Msg);
			IF idNode>=1 AND idNode<=MAX_LUXNUM THEN
				tmpIndex:=getGeolumenNodeByGeolumenId (idNode);
				IF(tmpIndex>0) THEN
					LuxGeolumenNodes[tmpIndex](feedbackState:=state); LuxGeolumenNodes[tmpIndex].updateFeedbackState();
				END_IF
			END_IF*)
		ELSIF  FIND(MsgRecBufferPtr^[ArrayPos].Msg,  '>' ) = 1 (* Isolo la sottostringa iniziale - > *) THEN
						MsgRecBufferPtr^[ArrayPos].MsgType := ECHO;
		ELSIF  FIND(MsgRecBufferPtr^[ArrayPos].Msg,  'Delete Operation Complete' ) = 1 (* Isolo la sottostringa iniziale - Delete Operation Complete *) THEN
						MsgRecBufferPtr^[ArrayPos].MsgType := NODE_DELETED;
	END_IF


	IF ArrayPos<MAX_ARRAY_MSG THEN
		ArrayPos:=ArrayPos+1;
	ELSE
		ArrayPos:=0;
	END_IF

	MsgRecBufferPtr^[ArrayPos].Msg:='';
	MsgRecBufferPtr^[ArrayPos].MsgType := COMPLETED;
	MsgRecBufferPtr^[ArrayPos].dwMacAdd:=0;
	(*MsgRecBufferPtr^[ArrayPos+1].Msg:='';
	MsgRecBufferPtr^[ArrayPos+1].MsgType := COMPLETED;
	MsgRecBufferPtr^[ArrayPos+1].dwMacAdd:=0;*)

END_IF;

(* clean buffer *)
ReceiveBufferPtr^.Index := 0;
FOR i:=0 TO 255 DO
	 ReceiveBufferPtr^.Data[i]:=16#00;
END_FOR;

(* conto i frame che ho ricevuto *)
contFrame:=contFrame+1;

END_IF;
END_ACTION
ACTION GetAndParseMessage2:
IF pReceiveStr = 0 THEN
	pReceiveStr := ADR(ReceiveBufferPtr^.Data);
END_IF

IF (ReceiveBufferPtr^.Index > 0 ) THEN

	(*gestione ricezione messaggi, consdierando eventuali spezzettamenti*)

	(*stringa ricevuta da seriale *)
	StringaDaSeriale :=  pReceiveStr^ ;

	IF DEBUG_SERIAL THEN
		logSerialInMessageRaw(StringaDaSeriale);
	END_IF

	(*posizione di CR+LF nella stringa ricevuta*)
	appoggioPosFullPrefix:=FIND(StringaDaSeriale,'$R$N');
	(*posizione di LF nella stringa ricevuta*)
	appoggioPosPartPrefix:=FIND(StringaDaSeriale,'$N');
	superatoAvanzo2:='';
	superatoAvanzo3:='';

	(*diagnostica: memorizzo dimensione max stringa da seriale e max dimensione di concatenamento tra tempString e stringa da seriale*)
	IF LEN(tempStringa)+LEN(StringaDaSeriale)>maxConcat THEN
		maxConcat:=LEN(tempStringa)+LEN(StringaDaSeriale);
	END_IF
	IF LEN(StringaDaSeriale) > maxStringaDaSerialeLength THEN
		maxStringaDaSerialeLength:=LEN(StringaDaSeriale);
	END_IF

	(*se c'è una terminazione completa => è un messaggio intero o la parte finale di un messaggio
		=> se ci sta in tempStringa lo concateno a tempStringa
	*)
	IF appoggioPosFullPrefix>0 AND appoggioPosFullPrefix+1 +LEN(tempStringa)<=255 THEN
		stringaSerialeCaso2:=StringaDaSeriale;
		appoggioCaso2:=LEFT(StringaDaSeriale,appoggioPosFullPrefix+1);
		IF(LEN(tempStringa)+LEN(appoggioCaso2))<=255 THEN
			tempStringaCaso2:=CONCAT(tempStringa,appoggioCaso2);
			superatoAvanzo2:=MID(StringaDaSeriale,LEN(StringaDaSeriale)-appoggioPosFullPrefix+1,appoggioPosFullPrefix+2);
		ELSE
			(*qui non dovrei mai arrivare...per sicurezza estrema*)
			caso2NonPotuto:=caso2NonPotuto+1;
		END_IF
		tempStringa:=tempStringaCaso2;

		(*per tenere come prima*)
		(*tempStringa:='';
		tempStringa :=CONCAT(tempStringa, StringaDaSeriale);*)

	(* altrimenti se c'è una terminazione parziale solo con CR =>
		=> se ci sta concateno in tempStringa
	*)
	ELSIF appoggioPosPartPrefix>0 AND appoggioPosPartPrefix +LEN(tempStringa)<=255 THEN
		stringaSerialeCaso3:=StringaDaSeriale;
		appoggioCaso3:=LEFT(StringaDaSeriale,appoggioPosPartPrefix);
		IF(LEN(tempStringa)+LEN(appoggioCaso3))<=255 THEN
			tempStringaCaso3:=CONCAT(tempStringa,appoggioCaso3);
			superatoAvanzo3:=MID(StringaDaSeriale,LEN(StringaDaSeriale)-appoggioPosPartPrefix,appoggioPosPartPrefix+1);
		ELSE
			caso3NonPotuto:=caso3NonPotuto+1;
		END_IF

		tempStringa:=tempStringaCaso3;
		(*per tenere come prima*)
		(*tempStringa:='';
		tempStringa :=CONCAT(tempStringa, StringaDaSeriale);*)

	(*se non ho né terminazione completa né parziale accodo in tempStringa se ci sta*)
	ELSIF (LEN(tempStringa)+LEN(StringaDaSeriale)<=255)   THEN
		tempStringa :=CONCAT(tempStringa, StringaDaSeriale);

	(*..altrimenti resetto tempStringa e prendo ciò che è arrivato. Non dovrei arrivare mai qui. *)
	ELSE
		LastSuperatoTime:=SYS.Time_CT_DT;
		superatoTEMPSTRINGA:=tempStringa;
		superatoSTRINGADASERIALE:=StringaDaSeriale;
		tempStringa:='';
		tempStringa :=CONCAT(tempStringa, StringaDaSeriale);
	END_IF

	(* QUI LOGICA DI PARSING *)
	(*trovo posizione di terminatore compleot in tempStringa*)
	tempBegin:=FIND(tempStringa,'$R$N');
	IF(tempBegin>0) THEN
		(* prendo solo parte sinistra: l'eccedenza a destra l'ho già nelle stringhe 'superatoAvanzo' e
		     lo considero alla fine dopo questo if *)
		LastMessage:=LEFT(tempStringa,tempBegin-1);
		tempStringa:='';

		(*
		(*rimosso non utile*)
		IF DEBUG_SERIAL THEN
			logSerialInMessage(LastMessage);
		END_IF*)

		MsgRecBuffer[ArrayPos].Msg:=LastMessage;
		LenghtStr:= LEN(MsgRecBuffer[ArrayPos].Msg);
		TrimStr1:=MID(MsgRecBuffer[ArrayPos].Msg, 3, 1); (*Isolo la sottostringa iniziale -  '#!#' *)

		(*se c'è l'inizio di un messaggio completo*)
		IF(SysStrCmp(TrimStr1, '#.#') = 0) THEN
			TrimStr1:=MID(MsgRecBuffer[ArrayPos].Msg, 7, 4); (*Isolo la sottostringa iniziale - REQAUTH*)
			TrimStr2:=MID(MsgRecBuffer[ArrayPos].Msg, 4, 32); (*Isolo la sottostringa finale - STS0*)

			IF (SysStrCmp(TrimStr1, 'REQAUTH') = 0 AND SysStrCmp(TrimStr2, 'STS0') = 0) THEN
				MsgRecBuffer[ArrayPos].MsgType := REQAUTH0;
				logRequestSTS0(MsgRecBuffer[ArrayPos].Msg);
				(*contSts0:=contSts0+1;*)
			ELSIF (SysStrCmp(TrimStr1, 'REQAUTH') = 0 AND SysStrCmp(TrimStr2, 'STS1') = 0) THEN
				MsgRecBuffer[ArrayPos].MsgType := REQAUTH1;
				(*contSts1:=contSts1+1;*)
			ELSE
				TrimNMEAS:=MID(MsgRecBuffer[ArrayPos].Msg, 6, 4); (* Isolo la sottostringa iniziale - NMEAS*)
				IF (SysStrCmp(TrimNMEAS, 'NMEAS;') = 0  AND   FIND(MsgRecBuffer[ArrayPos].Msg,  '#!#' ) > 0) THEN
					MsgRecBufferPtr^[ArrayPos].MsgType := DATAREC;
					(*identifico a quale nodo lux geolumen si riferisce e aggiorno stato*)
					parseNodeStatus(statusNodeMessage:=MsgRecBufferPtr^[ArrayPos].Msg);
					IF idNode>=1 AND idNode<=MAX_LUXNUM THEN
						tmpIndex:=getGeolumenNodeByGeolumenId (idNode);
						IF(tmpIndex>0 AND tmpIndex<=MAX_LUXNUM) THEN
							LuxGeolumenNodes[tmpIndex](feedbackState:=state); LuxGeolumenNodes[tmpIndex].updateFeedbackState();
						END_IF
					END_IF
				END_IF

				TrimNMEAS_Med:=MID(MsgRecBuffer[ArrayPos].Msg, 8, 4); (* Isolo la sottostringa iniziale - NMEASMED*)
				IF (SysStrCmp(TrimNMEAS_Med, 'NMEASMED') = 0  AND   FIND(MsgRecBuffer[ArrayPos].Msg,  '#!#' ) > 0) THEN
					MsgRecBufferPtr^[ArrayPos].MsgType := MED;
				END_IF
			END_IF

		ELSIF  FIND(MsgRecBufferPtr^[ArrayPos].Msg, ECHO_SET_LIGHT_ID_NODE_PREFIX[GEOLUMEN_COORD_VERSION] ) = 1 (* Isolo la sottostringa iniziale - >echo set *) THEN
			MsgRecBufferPtr^[ArrayPos].MsgType := ECHO;
			parseNodeEcho(echoNodeMessage:=MsgRecBufferPtr^[ArrayPos].Msg);
			IF echoset_IdNode>=1 AND echoset_IdNode<=MAX_LUXNUM THEN
				tmpIndex:=getGeolumenNodeByGeolumenId (echoset_IdNode);
				IF(tmpIndex>0 AND tmpIndex<=MAX_LUXNUM) THEN
					LuxGeolumenNodes[tmpIndex](echoCommandState:=echoCommandState); LuxGeolumenNodes[tmpIndex].updateEchoState();
				END_IF
			END_IF
		ELSIF  FIND(MsgRecBufferPtr^[ArrayPos].Msg,  '>' ) = 1 (* Isolo la sottostringa iniziale - > *)(*only v1*) THEN
						MsgRecBufferPtr^[ArrayPos].MsgType := ECHO;
		ELSIF  FIND(MsgRecBufferPtr^[ArrayPos].Msg,  'Delete Operation Complete' ) = 1 (* Isolo la sottostringa iniziale - Delete Operation Complete *) THEN
						MsgRecBufferPtr^[ArrayPos].MsgType := NODE_DELETED;
	END_IF


	IF LEN(appoggioCaso2) >0 THEN
		tempStringa:=superatoAvanzo2;
	ELSIF LEN(appoggioCaso3)>0 THEN
		tempStringa:=superatoAvanzo3;
	END_IF


	IF ArrayPos<MAX_ARRAY_MSG THEN
		ArrayPos:=ArrayPos+1;
	ELSE
		ArrayPos:=0;
	END_IF

	MsgRecBufferPtr^[ArrayPos].Msg:='';
	MsgRecBufferPtr^[ArrayPos].MsgType := COMPLETED;
	MsgRecBufferPtr^[ArrayPos].dwMacAdd:=0;

END_IF;

(* clean buffer *)
ReceiveBufferPtr^.Index := 0;
FOR i:=0 TO 255 DO
	 ReceiveBufferPtr^.Data[i]:=16#00;
END_FOR;

(* conto i frame che ho ricevuto *)
(*contFrame:=contFrame+1;*)

END_IF;
END_ACTION
ACTION luxRecall:
	FOR x:= 1 TO MAX_LUXNUM DO


		LuxElement[x].ID:=TabListLux[x].LuxNumber;
		ASTR[x].ID:=TabListLux[x].LuxNumber;

	END_FOR
END_ACTION
ACTION parseNodeEcho:
(*get node id - idn*)
echoset_idNodeStart:=FINDP(echoNodeMessage,ECHO_SET_LIGHT_ID_NODE_PREFIX[GEOLUMEN_COORD_VERSION],1);
echoset_partialStringNode:=DELETE(echoNodeMessage,echoset_idNodeStart+LEN(ECHO_SET_LIGHT_ID_NODE_PREFIX[GEOLUMEN_COORD_VERSION])-1,1);
echoset_posSeparator:=FINDP(echoset_partialStringNode, ECHO_SET_LIGHT_NODE_SEPARATOR[GEOLUMEN_COORD_VERSION],1);
echoset_idNode:=STRING_TO_WORD(MID(echoset_partialStringNode,echoset_posSeparator-1,1));

(*get node id - PW0*)
echoset_partialStringNode:=DELETE(echoset_partialStringNode,echoset_posSeparator,1);
echoset_idPw0Start:=FINDP(echoset_partialStringNode,SET_LIGHT_PW_SEPARATOR,1);
echoset_pwm0:=STRING_TO_WORD(MID(echoset_partialStringNode,echoset_idPw0Start-1,1));

(*get node id - PW1*)
echoset_partialStringNode:=DELETE(echoset_partialStringNode,echoset_idPw0Start,1);
echoset_idPw1Start:=FINDP(echoset_partialStringNode,SET_LIGHT_PW_SEPARATOR,1);
echoset_pwm1:=STRING_TO_WORD(MID(echoset_partialStringNode,echoset_idPw1Start-1,1));

(*get node id - PW2*)
echoset_partialStringNode:=DELETE(echoset_partialStringNode,echoset_idPw1Start,1);
echoset_pwm2:=STRING_TO_WORD(echoset_partialStringNode);

echoCommandState.id_Geolumen:=echoset_idNode;
echoCommandState.DimmValue_0:=echoset_pwm0;
echoCommandState.DimmValue_1:=echoset_pwm1;
echoCommandState.DimmValue_2:=echoset_pwm2;
END_ACTION
ACTION parseNodeStatus:
(*get node id - idn*)
idNodeStart:=FINDP(statusNodeMessage,ID_NODE_PREFIX,1);
partialStringNode:=DELETE(statusNodeMessage,idNodeStart+LEN(ID_NODE_PREFIX)-1,1);
posSeparator:=FINDP(partialStringNode, FIELD_SEPARATOR,1);
idNode:=STRING_TO_WORD(MID(partialStringNode,posSeparator-1,1));

(*get node id - PW0*)
idPw0Start:=FINDP(statusNodeMessage,PW0_PREFIX,1);
partialStringPW0:=DELETE(statusNodeMessage,idPw0Start+LEN(PW0_PREFIX)-1,1);
posSeparator:=FINDP(partialStringPW0, FIELD_SEPARATOR,1);
pwm0:=STRING_TO_WORD(MID(partialStringPW0,posSeparator-1,1));

(*get node id - PW1*)
idPw1Start:=FINDP(statusNodeMessage,PW1_PREFIX,1);
partialStringPW1:=DELETE(statusNodeMessage,idPw1Start+LEN(PW1_PREFIX)-1,1);
posSeparator:=FINDP(partialStringPW1, FIELD_SEPARATOR,1);
pwm1:=STRING_TO_WORD(MID(partialStringPW1,posSeparator-1,1));

(*get node id - PW2*)
idPw2Start:=FINDP(statusNodeMessage,PW2_PREFIX,1);
partialStringPW2:=DELETE(statusNodeMessage,idPw2Start+LEN(PW2_PREFIX)-1,1);
posSeparator:=FINDP(partialStringPW2, FIELD_SEPARATOR,1);
pwm2:=STRING_TO_WORD(MID(partialStringPW2,posSeparator-1,1));

(*get lamp current *)
idLampCurrentStart:=FINDP(statusNodeMessage,LAMP_CURRENT_PREFIX,1);
partialStringLampCurrent:=DELETE(statusNodeMessage,idLampCurrentStart+LEN(LAMP_CURRENT_PREFIX)-1,1);
posSeparator:=FINDP(partialStringLampCurrent, FIELD_SEPARATOR,1);
lampCurrent:=STRING_TO_WORD(MID(partialStringLampCurrent,posSeparator-1,1));

(*get lamp voltage*)
idLampVoltageStart:=FINDP(statusNodeMessage,LAMP_VOLTAGE_PREFIX,1);
partialStringLampVoltage:=DELETE(statusNodeMessage,idLampVoltageStart+LEN(LAMP_VOLTAGE_PREFIX)-1,1);
posSeparator:=FINDP(partialStringLampVoltage, FIELD_SEPARATOR,1);
LampVoltage:=STRING_TO_WORD(MID(partialStringLampVoltage,posSeparator-1,1));

(*get lamp power*)
idLampPowerStart:=FINDP(statusNodeMessage,LAMP_POWER_PREFIX,1);
partialStringLampPower:=DELETE(statusNodeMessage,idLampPowerStart+LEN(LAMP_POWER_PREFIX)-1,1);
posSeparator:=FINDP(partialStringLampPower, FIELD_SEPARATOR,1);
lampPower:=STRING_TO_WORD(MID(partialStringLampPower,posSeparator-1,1));


(*get PAR*)
idParCurrentStart:=FINDP(statusNodeMessage,PAR_PREFIX,1);
partialStringPar:=DELETE(statusNodeMessage,idParCurrentStart+LEN(PAR_PREFIX)-1,1);
posSeparator:=FINDP(partialStringPar, FIELD_SEPARATOR,1);
lastPar:=MID(partialStringPar,posSeparator-1,1);

(*get LQI*)
idLqiStart:=FINDP(statusNodeMessage,LQI_PREFIX,1);
partialStringLqi:=DELETE(statusNodeMessage,idLqiStart+LEN(LQI_PREFIX)-1,1);
posSeparator:=FINDP(partialStringLqi,FIELD_SEPARATOR,1);
lqiLast:=STRING_TO_WORD(MID(partialStringLqi,posSeparator-1,1));
IF(lqiLast > lqiMax) THEN lqiMax :=lqiLast; END_IF
IF(lqiLast < lqiMin) THEN lqiMin :=lqiLast; END_IF
IF countMsg<1000 THEN
	sumLqi:=sumLqi+lqiLast ;
	countMsg:=countMsg+1;
	lqiAvg:=REAL_TO_WORD(DWORD_TO_REAL(sumLqi)/DWORD_TO_REAL(countMsg));
ELSE
	countMsg:=1;
	sumLqi:=lqiLast;
	lqiAvg:=lqiLast;
END_IF

state.id_Geolumen:=idNode;
state.DimmValue_0:=pwm0;
state.DimmValue_1:=pwm1;
state.DimmValue_2:=pwm2;
state.LampCurrent:=lampCurrent;state.LampPower:=lampPower;state.LampVoltage:=lampVoltage;
state.lqiLast:=lqiLast;
state.lqiAvg:=lqiAvg;
state.lqiMax:=lqiMax;
state.lqiMin:=lqiMin;
state.lastPar:=lastPar;
END_ACTION
ACTION ReadID:
(* Ricerca tra i messaggi arrivati quali sono settati come DATAREC e quindi usa i dati per definire l'ID associato a quel lux e depositarlo nella struttura TabListLux *)

(*...per compabilità indicizzazione Renato...*)
counter:=ArrayPos-1;
IF(counter<0) THEN counter:=0; END_IF

